LIN {X 0,Y 431.431,Z 392.895,A -85,B 0,C 180,E1 -9540.932,E2 -9540.932} C_VEL
LIN {X 0,Y 431.488,Z 391.643,A -85,B 0,C 180,E1 -9541.866,E2 -9541.866} C_VEL
LIN {X 0,Y 431.805,Z 388.442,A -85,B 0,C 180,E1 -9543.264,E2 -9543.264} C_VEL
LIN {X 0,Y 431.906,Z 385.263,A -85,B 0,C 180,E1 -9544.198,E2 -9544.198} C_VEL
LIN {X 0,Y 432.129,Z 379.971,A -85,B 0,C 180,E1 -9545.365,E2 -9545.365} C_VEL
LIN {X 0,Y 432.279,Z 374.459,A -85,B 0,C 180,E1 -9546.299,E2 -9546.299} C_VEL
LIN {X 0,Y 432.336,Z 367.466,A -85,B 0,C 180,E1 -9547.221,E2 -9547.221} C_VEL
LIN {X 0,Y 432.6,Z 359.724,A -85,B 0,C 180,E1 -9548.018,E2 -9548.018} C_VEL
LIN {X 0,Y 432.755,Z 351.837,A -85,B 0,C 180,E1 -9548.638,E2 -9548.638} C_VEL
LIN {X 0,Y 432.779,Z 343.053,A -85,B 0,C 180,E1 -9549.168,E2 -9549.168} C_VEL
LIN {X 0,Y 431.838,Z 336.706,A -85,B 0,C 180,E1 -9549.483,E2 -9549.483} C_VEL
LIN {X 0,Y 431.977,Z 329.555,A -85,B 0,C 180,E1 -9552.534,E2 -9552.534} C_VEL
LIN {X 0,Y 431.962,Z 320.915,A -85,B 0,C 180,E1 -9556.274,E2 -9556.274} C_VEL
LIN {X 0,Y 432.057,Z 313.809,A -85,B 0,C 180,E1 -9559.36,E2 -9559.36} C_VEL
LIN {X 0,Y 432.075,Z 306.679,A -85,B 0,C 180,E1 -9562.471,E2 -9562.471} C_VEL
LIN {X 0,Y 432.147,Z 299.603,A -85,B 0,C 180,E1 -9565.527,E2 -9565.527} C_VEL
LIN {X 0,Y 432.259,Z 292.542,A -85,B 0,C 180,E1 -9568.601,E2 -9568.601} C_VEL
LIN {X 0,Y 432.354,Z 290.632,A -85,B 0,C 180,E1 -9569.452,E2 -9569.452} C_VEL
LIN {X 0,Y 432.31,Z 290.631,A -85,B 0,C 180,E1 -9572.442,E2 -9572.442} C_VEL
LIN {X 0,Y 432.33,Z 290.629,A -85,B 0,C 180,E1 -9575.817,E2 -9575.817} C_VEL
LIN {X 0,Y 432.323,Z 290.633,A -85,B 0,C 180,E1 -9578.711,E2 -9578.711} C_VEL
LIN {X 0,Y 432.313,Z 290.632,A -85,B 0,C 180,E1 -9581.797,E2 -9581.797} C_VEL
LIN {X 0,Y 432.326,Z 290.632,A -85,B 0,C 180,E1 -9584.346,E2 -9584.346} C_VEL
LIN {X 0,Y 432.312,Z 290.635,A -85,B 0,C 180,E1 -9587.014,E2 -9587.014} C_VEL
LIN {X 0,Y 432.333,Z 290.631,A -85,B 0,C 180,E1 -9589.818,E2 -9589.818} C_VEL
LIN {X 0,Y 432.307,Z 290.634,A -85,B 0,C 180,E1 -9593.022,E2 -9593.022} C_VEL
LIN {X 0,Y 432.35,Z 290.63,A -85,B 0,C 180,E1 -9595.995,E2 -9595.995} C_VEL
LIN {X 0,Y 432.385,Z 290.625,A -85,B 0,C 180,E1 -9599.743,E2 -9599.743} C_VEL
LIN {X 0,Y 432.39,Z 290.625,A -85,B 0,C 180,E1 -9603.371,E2 -9603.371} C_VEL
LIN {X 0,Y 432.36,Z 290.629,A -85,B 0,C 180,E1 -9606.023,E2 -9606.023} C_VEL
LIN {X 0,Y 432.339,Z 290.632,A -85,B 0,C 180,E1 -9609.045,E2 -9609.045} C_VEL
LIN {X 0,Y 432.366,Z 290.627,A -85,B 0,C 180,E1 -9612.011,E2 -9612.011} C_VEL
LIN {X 0,Y 432.383,Z 290.626,A -85,B 0,C 180,E1 -9614.926,E2 -9614.926} C_VEL
LIN {X 0,Y 432.446,Z 290.616,A -85,B 0,C 180,E1 -9617.803,E2 -9617.803} C_VEL
LIN {X 0,Y 432.451,Z 290.615,A -85,B 0,C 180,E1 -9621.589,E2 -9621.589} C_VEL
LIN {X 0,Y 432.567,Z 290.604,A -85,B 0,C 180,E1 -9624.406,E2 -9624.406} C_VEL
LIN {X 0,Y 432.582,Z 290.603,A -85,B 0,C 180,E1 -9628.138,E2 -9628.138} C_VEL
LIN {X 0,Y 432.597,Z 290.601,A -85,B 0,C 180,E1 -9630.119,E2 -9630.119} C_VEL
LIN {X 0,Y 432.548,Z 290.602,A -85,B 0,C 180,E1 -9632.794,E2 -9632.794} C_VEL
LIN {X 0,Y 432.337,Z 290.629,A -85,B 0,C 180,E1 -9634.194,E2 -9634.194} C_VEL
LIN {X 0,Y 431.716,Z 290.706,A -85,B 0,C 180,E1 -9634.973,E2 -9634.973} C_VEL
LIN {X 0,Y 428.929,Z 291.054,A -85,B 0,C 180,E1 -9636.239,E2 -9636.239} C_VEL
LIN {X 0,Y 426.54,Z 291.353,A -85,B 0,C 180,E1 -9637.261,E2 -9637.261} C_VEL
LIN {X 0,Y 425.497,Z 291.483,A -85,B 0,C 180,E1 -9638.049,E2 -9638.049} C_VEL
LIN {X 0,Y 425.404,Z 291.493,A -85,B 0,C 180,E1 -9638.317,E2 -9638.317} C_VEL
LIN {X 0,Y 425.337,Z 291.505,A -85,B 0,C 180,E1 -9641.436,E2 -9641.436} C_VEL
LIN {X 0,Y 425.336,Z 291.503,A -85,B 0,C 180,E1 -9644.35,E2 -9644.35} C_VEL
LIN {X 0,Y 425.33,Z 291.507,A -85,B 0,C 180,E1 -9647.303,E2 -9647.303} C_VEL
LIN {X 0,Y 425.284,Z 291.51,A -85,B 0,C 180,E1 -9650.306,E2 -9650.306} C_VEL
LIN {X 0,Y 425.296,Z 291.509,A -85,B 0,C 180,E1 -9653.366,E2 -9653.366} C_VEL
LIN {X 0,Y 425.338,Z 291.504,A -85,B 0,C 180,E1 -9656.845,E2 -9656.845} C_VEL
LIN {X 0,Y 425.308,Z 291.508,A -85,B 0,C 180,E1 -9659.718,E2 -9659.718} C_VEL
LIN {X 0,Y 425.275,Z 291.511,A -85,B 0,C 180,E1 -9663.049,E2 -9663.049} C_VEL
LIN {X 0,Y 425.276,Z 291.511,A -85,B 0,C 180,E1 -9665.93,E2 -9665.93} C_VEL
LIN {X 0,Y 425.295,Z 291.508,A -85,B 0,C 180,E1 -9669.046,E2 -9669.046} C_VEL
LIN {X 0,Y 425.267,Z 291.511,A -85,B 0,C 180,E1 -9672.654,E2 -9672.654} C_VEL
LIN {X 0,Y 425.253,Z 291.512,A -85,B 0,C 180,E1 -9676.045,E2 -9676.045} C_VEL
LIN {X 0,Y 425.249,Z 291.513,A -85,B 0,C 180,E1 -9678.621,E2 -9678.621} C_VEL
LIN {X 0,Y 425.274,Z 291.513,A -85,B 0,C 180,E1 -9681.101,E2 -9681.101} C_VEL
LIN {X 0,Y 425.288,Z 291.511,A -85,B 0,C 180,E1 -9684.665,E2 -9684.665} C_VEL
LIN {X 0,Y 425.325,Z 291.502,A -85,B 0,C 180,E1 -9688.08,E2 -9688.08} C_VEL
LIN {X 0,Y 425.41,Z 291.557,A -85,B 0,C 180,E1 -9689.302,E2 -9689.302} C_VEL
LIN {X 0,Y 425.439,Z 295.465,A -85,B 0,C 180,E1 -9691.378,E2 -9691.378} C_VEL
LIN {X 0,Y 425.168,Z 301.535,A -85,B 0,C 180,E1 -9694.548,E2 -9694.548} C_VEL
LIN {X 0,Y 424.965,Z 307.922,A -85,B 0,C 180,E1 -9697.838,E2 -9697.838} C_VEL
LIN {X 0,Y 424.857,Z 313.552,A -85,B 0,C 180,E1 -9700.682,E2 -9700.682} C_VEL
LIN {X 0,Y 424.689,Z 319.597,A -85,B 0,C 180,E1 -9703.703,E2 -9703.703} C_VEL
LIN {X 0,Y 424.581,Z 327.506,A -85,B 0,C 180,E1 -9707.586,E2 -9707.586} C_VEL
LIN {X 0,Y 424.422,Z 332.382,A -85,B 0,C 180,E1 -9709.898,E2 -9709.898} C_VEL
LIN {X 0,Y 425.912,Z 342.722,A -85,B 0,C 180,E1 -9710.444,E2 -9710.444} C_VEL
LIN {X 0,Y 426.109,Z 349.157,A -85,B 0,C 180,E1 -9710.867,E2 -9710.867} C_VEL
LIN {X 0,Y 425.799,Z 357.927,A -85,B 0,C 180,E1 -9711.578,E2 -9711.578} C_VEL
LIN {X 0,Y 425.5,Z 365.939,A -85,B 0,C 180,E1 -9712.408,E2 -9712.408} C_VEL
LIN {X 0,Y 425.269,Z 373.188,A -85,B 0,C 180,E1 -9713.358,E2 -9713.358} C_VEL
LIN {X 0,Y 425.072,Z 380.203,A -85,B 0,C 180,E1 -9714.546,E2 -9714.546} C_VEL
LIN {X 0,Y 424.872,Z 385.525,A -85,B 0,C 180,E1 -9715.732,E2 -9715.732} C_VEL
LIN {X 0,Y 424.62,Z 390.099,A -85,B 0,C 180,E1 -9717.155,E2 -9717.155} C_VEL
LIN {X 0,Y 424.439,Z 392.202,A -85,B 0,C 180,E1 -9718.103,E2 -9718.103} C_VEL
LIN {X 0,Y 424.384,Z 393.597,A -85,B 0,C 180,E1 -9719.052,E2 -9719.052} C_VEL
LIN {X 0,Y 424.397,Z 394.313,A -85,B 0,C 180,E1 -9720.001,E2 -9720.001} C_VEL
LIN {X 0,Y 424.439,Z 394.36,A -85,B 0,C 180,E1 -9720.95,E2 -9720.95} C_VEL
LIN {X 0,Y 424.516,Z 393.742,A -85,B 0,C 180,E1 -9721.899,E2 -9721.899} C_VEL
LIN {X 0,Y 424.66,Z 392.447,A -85,B 0,C 180,E1 -9722.847,E2 -9722.847} C_VEL
LIN {X 0,Y 424.926,Z 390.439,A -85,B 0,C 180,E1 -9723.795,E2 -9723.795} C_VEL
LIN {X 0,Y 425.187,Z 387.687,A -85,B 0,C 180,E1 -9724.742,E2 -9724.742} C_VEL
LIN {X 0,Y 425.583,Z 383.077,A -85,B 0,C 180,E1 -9725.925,E2 -9725.925} C_VEL
LIN {X 0,Y 425.972,Z 376.983,A -85,B 0,C 180,E1 -9727.109,E2 -9727.109} C_VEL
LIN {X 0,Y 426.429,Z 369.893,A -85,B 0,C 180,E1 -9728.171,E2 -9728.171} C_VEL
LIN {X 0,Y 426.984,Z 361.78,A -85,B 0,C 180,E1 -9729.116,E2 -9729.116} C_VEL
LIN {X 0,Y 427.458,Z 352.678,A -85,B 0,C 180,E1 -9729.942,E2 -9729.942} C_VEL
LIN {X 0,Y 427.53,Z 347.987,A -85,B 0,C 180,E1 -9730.299,E2 -9730.299} C_VEL
LIN {X 0,Y 425.577,Z 337.921,A -85,B 0,C 180,E1 -9731.009,E2 -9731.009} C_VEL
LIN {X 0,Y 424.97,Z 335.305,A -85,B 0,C 180,E1 -9731.206,E2 -9731.206} C_VEL
LIN {X 0,Y 425.162,Z 331.199,A -85,B 0,C 180,E1 -9733.382,E2 -9733.382} C_VEL
LIN {X 0,Y 425.431,Z 325.231,A -85,B 0,C 180,E1 -9736.635,E2 -9736.635} C_VEL
LIN {X 0,Y 425.776,Z 318.779,A -85,B 0,C 180,E1 -9740.283,E2 -9740.283} C_VEL
LIN {X 0,Y 426.086,Z 313.641,A -85,B 0,C 180,E1 -9743.321,E2 -9743.321} C_VEL
LIN {X 0,Y 426.534,Z 308.597,A -85,B 0,C 180,E1 -9746.417,E2 -9746.417} C_VEL
LIN {X 0,Y 426.992,Z 304.201,A -85,B 0,C 180,E1 -9749.267,E2 -9749.267} C_VEL
LIN {X 0,Y 427.019,Z 301.577,A -85,B 0,C 180,E1 -9751.148,E2 -9751.148} C_VEL
LIN {X 0,Y 426.838,Z 299.371,A -85,B 0,C 180,E1 -9752.913,E2 -9752.913} C_VEL
LIN {X 0,Y 426.407,Z 296.853,A -85,B 0,C 180,E1 -9755.231,E2 -9755.231} C_VEL
LIN {X 0,Y 425.993,Z 294.732,A -85,B 0,C 180,E1 -9757.636,E2 -9757.636} C_VEL
LIN {X 0,Y 425.623,Z 292.959,A -85,B 0,C 180,E1 -9760.574,E2 -9760.574} C_VEL
LIN {X 0,Y 425.422,Z 292.31,A -85,B 0,C 180,E1 -9763.374,E2 -9763.374} C_VEL
LIN {X 0,Y 425.543,Z 292.781,A -85,B 0,C 180,E1 -9766.08,E2 -9766.08} C_VEL
LIN {X 0,Y 425.84,Z 293.804,A -85,B 0,C 180,E1 -9767.961,E2 -9767.961} C_VEL
LIN {X 0,Y 426.327,Z 295.602,A -85,B 0,C 180,E1 -9769.99,E2 -9769.99} C_VEL
LIN {X 0,Y 427.12,Z 298.823,A -85,B 0,C 180,E1 -9772.496,E2 -9772.496} C_VEL
LIN {X 0,Y 428.239,Z 303.443,A -85,B 0,C 180,E1 -9775.143,E2 -9775.143} C_VEL
LIN {X 0,Y 429.35,Z 308.119,A -85,B 0,C 180,E1 -9777.304,E2 -9777.304} C_VEL
LIN {X 0,Y 430.605,Z 314.841,A -85,B 0,C 180,E1 -9779.887,E2 -9779.887} C_VEL
LIN {X 0,Y 430.728,Z 317.29,A -85,B 0,C 180,E1 -9780.692,E2 -9780.692} C_VEL
LIN {X 0,Y 429.254,Z 326.071,A -85,B 0,C 180,E1 -9783.24,E2 -9783.24} C_VEL
LIN {X 0,Y 427.548,Z 339.217,A -85,B 0,C 180,E1 -9786.764,E2 -9786.764} C_VEL
LIN {X 0,Y 426.625,Z 349.188,A -85,B 0,C 180,E1 -9789.257,E2 -9789.257} C_VEL
LIN {X 0,Y 425.685,Z 363.777,A -85,B 0,C 180,E1 -9792.712,E2 -9792.712} C_VEL
LIN {X 0,Y 425.548,Z 366.714,A -85,B 0,C 180,E1 -9793.388,E2 -9793.388} C_VEL
LIN {X 0,Y 427.239,Z 380.58,A -85,B 0,C 180,E1 -9793.883,E2 -9793.883} C_VEL
LIN {X 0,Y 427.862,Z 392.817,A -85,B 0,C 180,E1 -9794.458,E2 -9794.458} C_VEL
LIN {X 0,Y 427.224,Z 405.62,A -85,B 0,C 180,E1 -9795.227,E2 -9795.227} C_VEL
LIN {X 0,Y 426.563,Z 416.33,A -85,B 0,C 180,E1 -9796.057,E2 -9796.057} C_VEL
LIN {X 0,Y 426.089,Z 426.068,A -85,B 0,C 180,E1 -9796.996,E2 -9796.996} C_VEL
LIN {X 0,Y 425.42,Z 435.337,A -85,B 0,C 180,E1 -9798.083,E2 -9798.083} C_VEL
LIN {X 0,Y 424.995,Z 443.71,A -85,B 0,C 180,E1 -9799.278,E2 -9799.278} C_VEL
LIN {X 0,Y 424.666,Z 451.921,A -85,B 0,C 180,E1 -9800.714,E2 -9800.714} C_VEL
LIN {X 0,Y 424.5,Z 457.482,A -85,B 0,C 180,E1 -9801.91,E2 -9801.91} C_VEL
LIN {X 0,Y 424.376,Z 463.56,A -85,B 0,C 180,E1 -9803.544,E2 -9803.544} C_VEL
LIN {X 0,Y 424.29,Z 468.247,A -85,B 0,C 180,E1 -9805.249,E2 -9805.249} C_VEL
LIN {X 0,Y 424.391,Z 470.225,A -85,B 0,C 180,E1 -9806.202,E2 -9806.202} C_VEL
LIN {X 0,Y 424.431,Z 471.7,A -85,B 0,C 180,E1 -9807.153,E2 -9807.153} C_VEL
LIN {X 0,Y 424.379,Z 472.748,A -85,B 0,C 180,E1 -9808.102,E2 -9808.102} C_VEL
LIN {X 0,Y 424.299,Z 473.383,A -85,B 0,C 180,E1 -9809.051,E2 -9809.051} C_VEL
LIN {X 0,Y 424.292,Z 473.558,A -85,B 0,C 180,E1 -9810,E2 -9810} C_VEL
LIN {X 0,Y 424.297,Z 473.314,A -85,B 0,C 180,E1 -9810.949,E2 -9810.949} C_VEL
LIN {X 0,Y 424.378,Z 472.67,A -85,B 0,C 180,E1 -9811.898,E2 -9811.898} C_VEL
LIN {X 0,Y 424.5,Z 471.576,A -85,B 0,C 180,E1 -9812.847,E2 -9812.847} C_VEL
LIN {X 0,Y 424.31,Z 469.054,A -85,B 0,C 180,E1 -9814.275,E2 -9814.275} C_VEL
LIN {X 0,Y 424.379,Z 465.475,A -85,B 0,C 180,E1 -9815.703,E2 -9815.703} C_VEL
LIN {X 0,Y 424.433,Z 460.7,A -85,B 0,C 180,E1 -9817.134,E2 -9817.134} C_VEL
LIN {X 0,Y 424.543,Z 454.589,A -85,B 0,C 180,E1 -9818.568,E2 -9818.568} C_VEL
LIN {X 0,Y 424.774,Z 446.92,A -85,B 0,C 180,E1 -9820.005,E2 -9820.005} C_VEL
LIN {X 0,Y 425.172,Z 438.998,A -85,B 0,C 180,E1 -9821.199,E2 -9821.199} C_VEL
LIN {X 0,Y 425.61,Z 430.347,A -85,B 0,C 180,E1 -9822.275,E2 -9822.275} C_VEL
LIN {X 0,Y 425.952,Z 422.768,A -85,B 0,C 180,E1 -9823.069,E2 -9823.069} C_VEL
LIN {X 0,Y 426.519,Z 411.011,A -85,B 0,C 180,E1 -9824.066,E2 -9824.066} C_VEL
LIN {X 0,Y 427.09,Z 399.322,A -85,B 0,C 180,E1 -9824.838,E2 -9824.838} C_VEL
LIN {X 0,Y 427.203,Z 388.532,A -85,B 0,C 180,E1 -9825.383,E2 -9825.383} C_VEL
LIN {X 0,Y 426,Z 375.127,A -85,B 0,C 180,E1 -9825.888,E2 -9825.888} C_VEL
LIN {X 0,Y 425.312,Z 367.811,A -85,B 0,C 180,E1 -9826.099,E2 -9826.099} C_VEL
LIN {X 0,Y 426.031,Z 354.032,A -85,B 0,C 180,E1 -9829.265,E2 -9829.265} C_VEL
LIN {X 0,Y 427.055,Z 339.899,A -85,B 0,C 180,E1 -9832.553,E2 -9832.553} C_VEL
LIN {X 0,Y 428.279,Z 325.124,A -85,B 0,C 180,E1 -9836.052,E2 -9836.052} C_VEL
LIN {X 0,Y 429.459,Z 312.388,A -85,B 0,C 180,E1 -9839.134,E2 -9839.134} C_VEL
LIN {X 0,Y 428.62,Z 306.988,A -85,B 0,C 180,E1 -9840.551,E2 -9840.551} C_VEL
LIN {X 0,Y 425.673,Z 293.201,A -85,B 0,C 180,E1 -9844.358,E2 -9844.358} C_VEL
LIN {X 0,Y 425.309,Z 291.509,A -85,B 0,C 180,E1 -9844.858,E2 -9844.858} C_VEL
LIN {X 0,Y 425.284,Z 291.512,A -85,B 0,C 180,E1 -9847.694,E2 -9847.694} C_VEL
LIN {X 0,Y 425.285,Z 291.513,A -85,B 0,C 180,E1 -9850.52,E2 -9850.52} C_VEL
LIN {X 0,Y 425.263,Z 291.512,A -85,B 0,C 180,E1 -9853.35,E2 -9853.35} C_VEL
LIN {X 0,Y 425.263,Z 291.512,A -85,B 0,C 180,E1 -9856.649,E2 -9856.649} C_VEL
LIN {X 0,Y 425.295,Z 291.508,A -85,B 0,C 180,E1 -9859.873,E2 -9859.873} C_VEL
LIN {X 0,Y 425.284,Z 291.511,A -85,B 0,C 180,E1 -9862.488,E2 -9862.488} C_VEL
LIN {X 0,Y 425.311,Z 291.511,A -85,B 0,C 180,E1 -9865.817,E2 -9865.817} C_VEL
LIN {X 0,Y 425.288,Z 291.514,A -85,B 0,C 180,E1 -9869.24,E2 -9869.24} C_VEL
LIN {X 0,Y 425.311,Z 291.731,A -85,B 0,C 180,E1 -9870.008,E2 -9870.008} C_VEL
LIN {X 0,Y 425.767,Z 295.291,A -85,B 0,C 180,E1 -9871.399,E2 -9871.399} C_VEL
LIN {X 0,Y 425.635,Z 303.415,A -85,B 0,C 180,E1 -9874.575,E2 -9874.575} C_VEL
LIN {X 0,Y 425.538,Z 312.26,A -85,B 0,C 180,E1 -9878.185,E2 -9878.185} C_VEL
LIN {X 0,Y 425.438,Z 319.451,A -85,B 0,C 180,E1 -9881.207,E2 -9881.207} C_VEL
LIN {X 0,Y 425.368,Z 326.466,A -85,B 0,C 180,E1 -9884.179,E2 -9884.179} C_VEL
LIN {X 0,Y 425.402,Z 335.436,A -85,B 0,C 180,E1 -9888.081,E2 -9888.081} C_VEL
LIN {X 0,Y 425.301,Z 339.67,A -85,B 0,C 180,E1 -9889.917,E2 -9889.917} C_VEL
LIN {X 0,Y 426.723,Z 347.144,A -85,B 0,C 180,E1 -9890.34,E2 -9890.34} C_VEL
LIN {X 0,Y 426.45,Z 356.821,A -85,B 0,C 180,E1 -9890.991,E2 -9890.991} C_VEL
LIN {X 0,Y 426.13,Z 365.402,A -85,B 0,C 180,E1 -9891.785,E2 -9891.785} C_VEL
LIN {X 0,Y 425.771,Z 372.676,A -85,B 0,C 180,E1 -9892.649,E2 -9892.649} C_VEL
LIN {X 0,Y 425.624,Z 378.737,A -85,B 0,C 180,E1 -9893.599,E2 -9893.599} C_VEL
LIN {X 0,Y 425.31,Z 383.556,A -85,B 0,C 180,E1 -9894.547,E2 -9894.547} C_VEL
LIN {X 0,Y 425.194,Z 388.08,A -85,B 0,C 180,E1 -9895.733,E2 -9895.733} C_VEL
LIN {X 0,Y 424.935,Z 390.704,A -85,B 0,C 180,E1 -9896.68,E2 -9896.68} C_VEL
LIN {X 0,Y 424.63,Z 391.791,A -85,B 0,C 180,E1 -9897.153,E2 -9897.153} C_VEL
LIN {X 0,Y 424.489,Z 393.276,A -85,B 0,C 180,E1 -9898.101,E2 -9898.101} C_VEL
LIN {X 0,Y 424.415,Z 394.045,A -85,B 0,C 180,E1 -9899.05,E2 -9899.05} C_VEL
LIN {X 0,Y 424.373,Z 394.123,A -85,B 0,C 180,E1 -9899.999,E2 -9899.999} C_VEL
LIN {X 0,Y 424.368,Z 393.517,A -85,B 0,C 180,E1 -9900.948,E2 -9900.948} C_VEL
LIN {X 0,Y 424.504,Z 391.341,A -85,B 0,C 180,E1 -9902.371,E2 -9902.371} C_VEL
LIN {X 0,Y 424.748,Z 388.935,A -85,B 0,C 180,E1 -9903.319,E2 -9903.319} C_VEL
LIN {X 0,Y 424.981,Z 383.756,A -85,B 0,C 180,E1 -9904.742,E2 -9904.742} C_VEL
LIN {X 0,Y 425.155,Z 377.656,A -85,B 0,C 180,E1 -9905.929,E2 -9905.929} C_VEL
LIN {X 0,Y 425.23,Z 370.847,A -85,B 0,C 180,E1 -9906.95,E2 -9906.95} C_VEL
LIN {X 0,Y 425.455,Z 363.083,A -85,B 0,C 180,E1 -9907.831,E2 -9907.831} C_VEL
LIN {X 0,Y 425.632,Z 355.043,A -85,B 0,C 180,E1 -9908.545,E2 -9908.545} C_VEL
LIN {X 0,Y 425.859,Z 345.965,A -85,B 0,C 180,E1 -9909.138,E2 -9909.138} C_VEL
LIN {X 0,Y 424.8,Z 337.288,A -85,B 0,C 180,E1 -9909.582,E2 -9909.582} C_VEL
LIN {X 0,Y 424.931,Z 330.165,A -85,B 0,C 180,E1 -9912.627,E2 -9912.627} C_VEL
LIN {X 0,Y 424.917,Z 321.461,A -85,B 0,C 180,E1 -9916.401,E2 -9916.401} C_VEL
LIN {X 0,Y 425.025,Z 314.285,A -85,B 0,C 180,E1 -9919.52,E2 -9919.52} C_VEL
LIN {X 0,Y 425.033,Z 306.667,A -85,B 0,C 180,E1 -9922.864,E2 -9922.864} C_VEL
LIN {X 0,Y 425.134,Z 299.493,A -85,B 0,C 180,E1 -9925.98,E2 -9925.98} C_VEL
LIN {X 0,Y 425.335,Z 291.506,A -85,B 0,C 180,E1 -9929.47,E2 -9929.47} C_VEL
LIN {X 0,Y 425.262,Z 291.513,A -85,B 0,C 180,E1 -9933.048,E2 -9933.048} C_VEL
LIN {X 0,Y 425.274,Z 291.508,A -85,B 0,C 180,E1 -9935.927,E2 -9935.927} C_VEL
LIN {X 0,Y 425.258,Z 291.516,A -85,B 0,C 180,E1 -9939.036,E2 -9939.036} C_VEL
LIN {X 0,Y 425.262,Z 291.513,A -85,B 0,C 180,E1 -9942.652,E2 -9942.652} C_VEL
LIN {X 0,Y 425.254,Z 291.512,A -85,B 0,C 180,E1 -9946.043,E2 -9946.043} C_VEL
LIN {X 0,Y 425.267,Z 291.515,A -85,B 0,C 180,E1 -9948.62,E2 -9948.62} C_VEL
LIN {X 0,Y 425.307,Z 291.506,A -85,B 0,C 180,E1 -9951.102,E2 -9951.102} C_VEL
LIN {X 0,Y 425.292,Z 291.509,A -85,B 0,C 180,E1 -9954.663,E2 -9954.663} C_VEL
LIN {X 0,Y 425.263,Z 291.513,A -85,B 0,C 180,E1 -9958.073,E2 -9958.073} C_VEL
LIN {X 0,Y 425.328,Z 291.505,A -85,B 0,C 180,E1 -9961.367,E2 -9961.367} C_VEL
LIN {X 0,Y 425.285,Z 291.51,A -85,B 0,C 180,E1 -9964.554,E2 -9964.554} C_VEL
LIN {X 0,Y 425.277,Z 291.51,A -85,B 0,C 180,E1 -9967.661,E2 -9967.661} C_VEL
LIN {X 0,Y 425.351,Z 291.504,A -85,B 0,C 180,E1 -9970.703,E2 -9970.703} C_VEL
LIN {X 0,Y 425.377,Z 291.498,A -85,B 0,C 180,E1 -9973.688,E2 -9973.688} C_VEL
LIN {X 0,Y 425.399,Z 291.494,A -85,B 0,C 180,E1 -9977.598,E2 -9977.598} C_VEL
LIN {X 0,Y 425.395,Z 291.494,A -85,B 0,C 180,E1 -9981.449,E2 -9981.449} C_VEL
LIN {X 0,Y 425.521,Z 291.483,A -85,B 0,C 180,E1 -9984.313,E2 -9984.313} C_VEL
LIN {X 0,Y 425.552,Z 291.479,A -85,B 0,C 180,E1 -9988.107,E2 -9988.107} C_VEL
LIN {X 0,Y 425.577,Z 291.477,A -85,B 0,C 180,E1 -9990,E2 -9990} C_VEL
LIN {X 0,Y 425.504,Z 291.479,A -85,B 0,C 180,E1 -9992.84,E2 -9992.84} C_VEL
LIN {X 0,Y 425.521,Z 291.483,A -85,B 0,C 180,E1 -9995.687,E2 -9995.687} C_VEL
LIN {X 0,Y 425.404,Z 291.493,A -85,B 0,C 180,E1 -9998.317,E2 -9998.317} C_VEL
LIN {X 0,Y 424.702,Z 291.582,A -85,B 0,C 180,E1 -9999.106,E2 -9999.106} C_VEL
LIN {X 0,Y 421.799,Z 291.942,A -85,B 0,C 180,E1 -10000.389,E2 -10000.389} C_VEL
LIN {X 0,Y 419.386,Z 292.246,A -85,B 0,C 180,E1 -10001.425,E2 -10001.425} C_VEL
LIN {X 0,Y 418.391,Z 292.367,A -85,B 0,C 180,E1 -10002.225,E2 -10002.225} C_VEL
LIN {X 0,Y 418.331,Z 292.374,A -85,B 0,C 180,E1 -10002.496,E2 -10002.496} C_VEL
LIN {X 0,Y 418.29,Z 292.382,A -85,B 0,C 180,E1 -10005.595,E2 -10005.595} C_VEL
LIN {X 0,Y 418.272,Z 292.382,A -85,B 0,C 180,E1 -10008.617,E2 -10008.617} C_VEL
LIN {X 0,Y 418.223,Z 292.389,A -85,B 0,C 180,E1 -10011.697,E2 -10011.697} C_VEL
LIN {X 0,Y 418.273,Z 292.384,A -85,B 0,C 180,E1 -10014.865,E2 -10014.865} C_VEL
LIN {X 0,Y 418.285,Z 292.382,A -85,B 0,C 180,E1 -10018.064,E2 -10018.064} C_VEL
LIN {X 0,Y 418.211,Z 292.391,A -85,B 0,C 180,E1 -10021.396,E2 -10021.396} C_VEL
LIN {X 0,Y 418.257,Z 292.385,A -85,B 0,C 180,E1 -10024.581,E2 -10024.581} C_VEL
LIN {X 0,Y 418.226,Z 292.389,A -85,B 0,C 180,E1 -10027.836,E2 -10027.836} C_VEL
LIN {X 0,Y 418.215,Z 292.39,A -85,B 0,C 180,E1 -10030.949,E2 -10030.949} C_VEL
LIN {X 0,Y 418.202,Z 292.391,A -85,B 0,C 180,E1 -10033.731,E2 -10033.731} C_VEL
LIN {X 0,Y 418.199,Z 292.391,A -85,B 0,C 180,E1 -10036.45,E2 -10036.45} C_VEL
LIN {X 0,Y 418.202,Z 292.394,A -85,B 0,C 180,E1 -10039.134,E2 -10039.134} C_VEL
LIN {X 0,Y 418.231,Z 292.39,A -85,B 0,C 180,E1 -10042.777,E2 -10042.777} C_VEL
LIN {X 0,Y 418.229,Z 292.387,A -85,B 0,C 180,E1 -10046.323,E2 -10046.323} C_VEL
LIN {X 0,Y 418.383,Z 292.437,A -85,B 0,C 180,E1 -10049.249,E2 -10049.249} C_VEL
LIN {X 0,Y 418.411,Z 296.46,A -85,B 0,C 180,E1 -10051.401,E2 -10051.401} C_VEL
LIN {X 0,Y 418.119,Z 302.556,A -85,B 0,C 180,E1 -10054.622,E2 -10054.622} C_VEL
LIN {X 0,Y 417.893,Z 309.625,A -85,B 0,C 180,E1 -10058.287,E2 -10058.287} C_VEL
LIN {X 0,Y 417.719,Z 315.644,A -85,B 0,C 180,E1 -10061.359,E2 -10061.359} C_VEL
LIN {X 0,Y 417.577,Z 321.653,A -85,B 0,C 180,E1 -10064.38,E2 -10064.38} C_VEL
LIN {X 0,Y 417.504,Z 327.987,A -85,B 0,C 180,E1 -10067.512,E2 -10067.512} C_VEL
LIN {X 0,Y 417.384,Z 332.795,A -85,B 0,C 180,E1 -10069.757,E2 -10069.757} C_VEL
LIN {X 0,Y 418.933,Z 343.651,A -85,B 0,C 180,E1 -10070.344,E2 -10070.344} C_VEL
LIN {X 0,Y 419.049,Z 350.807,A -85,B 0,C 180,E1 -10070.833,E2 -10070.833} C_VEL
LIN {X 0,Y 418.701,Z 360.518,A -85,B 0,C 180,E1 -10071.678,E2 -10071.678} C_VEL
LIN {X 0,Y 418.36,Z 369.233,A -85,B 0,C 180,E1 -10072.668,E2 -10072.668} C_VEL
LIN {X 0,Y 418.173,Z 376.491,A -85,B 0,C 180,E1 -10073.73,E2 -10073.73} C_VEL
LIN {X 0,Y 417.976,Z 382.872,A -85,B 0,C 180,E1 -10074.937,E2 -10074.937} C_VEL
LIN {X 0,Y 417.711,Z 387.709,A -85,B 0,C 180,E1 -10076.142,E2 -10076.142} C_VEL
LIN {X 0,Y 417.547,Z 390.617,A -85,B 0,C 180,E1 -10077.107,E2 -10077.107} C_VEL
LIN {X 0,Y 417.385,Z 392.775,A -85,B 0,C 180,E1 -10078.071,E2 -10078.071} C_VEL
LIN {X 0,Y 417.321,Z 394.228,A -85,B 0,C 180,E1 -10079.036,E2 -10079.036} C_VEL
LIN {X 0,Y 417.331,Z 394.998,A -85,B 0,C 180,E1 -10080.001,E2 -10080.001} C_VEL
LIN {X 0,Y 417.38,Z 395.098,A -85,B 0,C 180,E1 -10080.966,E2 -10080.966} C_VEL
LIN {X 0,Y 417.465,Z 394.529,A -85,B 0,C 180,E1 -10081.931,E2 -10081.931} C_VEL
LIN {X 0,Y 417.619,Z 393.285,A -85,B 0,C 180,E1 -10082.895,E2 -10082.895} C_VEL
LIN {X 0,Y 418.182,Z 390.079,A -85,B 0,C 180,E1 -10084.338,E2 -10084.338} C_VEL
LIN {X 0,Y 418.309,Z 387.039,A -85,B 0,C 180,E1 -10085.303,E2 -10085.303} C_VEL
LIN {X 0,Y 418.74,Z 382,A -85,B 0,C 180,E1 -10086.506,E2 -10086.506} C_VEL
LIN {X 0,Y 419.212,Z 375.354,A -85,B 0,C 180,E1 -10087.709,E2 -10087.709} C_VEL
LIN {X 0,Y 419.705,Z 368.559,A -85,B 0,C 180,E1 -10088.669,E2 -10088.669} C_VEL
LIN {X 0,Y 420.316,Z 359.904,A -85,B 0,C 180,E1 -10089.627,E2 -10089.627} C_VEL
LIN {X 0,Y 420.8,Z 350.076,A -85,B 0,C 180,E1 -10090.466,E2 -10090.466} C_VEL
LIN {X 0,Y 419.383,Z 341.712,A -85,B 0,C 180,E1 -10091.112,E2 -10091.112} C_VEL
LIN {X 0,Y 417.995,Z 335.834,A -85,B 0,C 180,E1 -10091.518,E2 -10091.518} C_VEL
LIN {X 0,Y 418.167,Z 331.965,A -85,B 0,C 180,E1 -10093.61,E2 -10093.61} C_VEL
LIN {X 0,Y 418.443,Z 326.227,A -85,B 0,C 180,E1 -10096.793,E2 -10096.793} C_VEL
LIN {X 0,Y 418.777,Z 320.686,A -85,B 0,C 180,E1 -10099.981,E2 -10099.981} C_VEL
LIN {X 0,Y 419.081,Z 316.104,A -85,B 0,C 180,E1 -10102.727,E2 -10102.727} C_VEL
LIN {X 0,Y 419.507,Z 311.197,A -85,B 0,C 180,E1 -10105.823,E2 -10105.823} C_VEL
LIN {X 0,Y 420.078,Z 306.336,A -85,B 0,C 180,E1 -10109.025,E2 -10109.025} C_VEL
LIN {X 0,Y 420.14,Z 303.104,A -85,B 0,C 180,E1 -10111.447,E2 -10111.447} C_VEL
LIN {X 0,Y 419.893,Z 300.675,A -85,B 0,C 180,E1 -10113.529,E2 -10113.529} C_VEL
LIN {X 0,Y 419.454,Z 297.869,A -85,B 0,C 180,E1 -10116.462,E2 -10116.462} C_VEL
LIN {X 0,Y 419.013,Z 295.785,A -85,B 0,C 180,E1 -10119.597,E2 -10119.597} C_VEL
LIN {X 0,Y 418.808,Z 294.887,A -85,B 0,C 180,E1 -10122.408,E2 -10122.408} C_VEL
LIN {X 0,Y 418.845,Z 295.057,A -85,B 0,C 180,E1 -10125.191,E2 -10125.191} C_VEL
LIN {X 0,Y 419.227,Z 296.359,A -85,B 0,C 180,E1 -10127.889,E2 -10127.889} C_VEL
LIN {X 0,Y 419.838,Z 298.756,A -85,B 0,C 180,E1 -10130.497,E2 -10130.497} C_VEL
LIN {X 0,Y 420.792,Z 302.652,A -85,B 0,C 180,E1 -10133.293,E2 -10133.293} C_VEL
LIN {X 0,Y 421.748,Z 306.604,A -85,B 0,C 180,E1 -10135.488,E2 -10135.488} C_VEL
LIN {X 0,Y 422.951,Z 312.007,A -85,B 0,C 180,E1 -10137.936,E2 -10137.936} C_VEL
LIN {X 0,Y 423.927,Z 317.911,A -85,B 0,C 180,E1 -10140.175,E2 -10140.175} C_VEL
LIN {X 0,Y 423.573,Z 321.255,A -85,B 0,C 180,E1 -10141.238,E2 -10141.238} C_VEL
LIN {X 0,Y 421.478,Z 333.704,A -85,B 0,C 180,E1 -10144.836,E2 -10144.836} C_VEL
LIN {X 0,Y 419.979,Z 347.243,A -85,B 0,C 180,E1 -10148.398,E2 -10148.398} C_VEL
LIN {X 0,Y 418.819,Z 361.565,A -85,B 0,C 180,E1 -10151.914,E2 -10151.914} C_VEL
LIN {X 0,Y 418.588,Z 366.57,A -85,B 0,C 180,E1 -10153.073,E2 -10153.073} C_VEL
LIN {X 0,Y 420.337,Z 379.858,A -85,B 0,C 180,E1 -10153.565,E2 -10153.565} C_VEL
LIN {X 0,Y 421.02,Z 392.898,A -85,B 0,C 180,E1 -10154.199,E2 -10154.199} C_VEL
LIN {X 0,Y 420.37,Z 405.488,A -85,B 0,C 180,E1 -10154.981,E2 -10154.981} C_VEL
LIN {X 0,Y 419.636,Z 416.066,A -85,B 0,C 180,E1 -10155.822,E2 -10155.822} C_VEL
LIN {X 0,Y 419.08,Z 426.423,A -85,B 0,C 180,E1 -10156.856,E2 -10156.856} C_VEL
LIN {X 0,Y 418.336,Z 436.715,A -85,B 0,C 180,E1 -10158.124,E2 -10158.124} C_VEL
LIN {X 0,Y 417.867,Z 444.741,A -85,B 0,C 180,E1 -10159.338,E2 -10159.338} C_VEL
LIN {X 0,Y 417.557,Z 452.572,A -85,B 0,C 180,E1 -10160.799,E2 -10160.799} C_VEL
LIN {X 0,Y 417.362,Z 458.86,A -85,B 0,C 180,E1 -10162.258,E2 -10162.258} C_VEL
LIN {X 0,Y 417.273,Z 463.42,A -85,B 0,C 180,E1 -10163.58,E2 -10163.58} C_VEL
LIN {X 0,Y 417.222,Z 467.638,A -85,B 0,C 180,E1 -10165.169,E2 -10165.169} C_VEL
LIN {X 0,Y 417.293,Z 469.593,A -85,B 0,C 180,E1 -10166.137,E2 -10166.137} C_VEL
LIN {X 0,Y 417.355,Z 471.057,A -85,B 0,C 180,E1 -10167.104,E2 -10167.104} C_VEL
LIN {X 0,Y 417.326,Z 472.098,A -85,B 0,C 180,E1 -10168.07,E2 -10168.07} C_VEL
LIN {X 0,Y 417.242,Z 472.713,A -85,B 0,C 180,E1 -10169.035,E2 -10169.035} C_VEL
LIN {X 0,Y 417.231,Z 472.867,A -85,B 0,C 180,E1 -10170,E2 -10170} C_VEL
LIN {X 0,Y 417.24,Z 472.61,A -85,B 0,C 180,E1 -10170.965,E2 -10170.965} C_VEL
LIN {X 0,Y 417.327,Z 471.952,A -85,B 0,C 180,E1 -10171.93,E2 -10171.93} C_VEL
LIN {X 0,Y 417.431,Z 470.821,A -85,B 0,C 180,E1 -10172.895,E2 -10172.895} C_VEL
LIN {X 0,Y 417.244,Z 468.259,A -85,B 0,C 180,E1 -10174.347,E2 -10174.347} C_VEL
LIN {X 0,Y 417.297,Z 464.631,A -85,B 0,C 180,E1 -10175.8,E2 -10175.8} C_VEL
LIN {X 0,Y 417.358,Z 459.8,A -85,B 0,C 180,E1 -10177.256,E2 -10177.256} C_VEL
LIN {X 0,Y 417.478,Z 453.623,A -85,B 0,C 180,E1 -10178.714,E2 -10178.714} C_VEL
LIN {X 0,Y 417.715,Z 445.835,A -85,B 0,C 180,E1 -10180.175,E2 -10180.175} C_VEL
LIN {X 0,Y 418.162,Z 437.807,A -85,B 0,C 180,E1 -10181.39,E2 -10181.39} C_VEL
LIN {X 0,Y 418.667,Z 429.038,A -85,B 0,C 180,E1 -10182.482,E2 -10182.482} C_VEL
LIN {X 0,Y 419.14,Z 418.234,A -85,B 0,C 180,E1 -10183.577,E2 -10183.577} C_VEL
LIN {X 0,Y 419.641,Z 407.646,A -85,B 0,C 180,E1 -10184.426,E2 -10184.426} C_VEL
LIN {X 0,Y 420.234,Z 394.959,A -85,B 0,C 180,E1 -10185.21,E2 -10185.21} C_VEL
LIN {X 0,Y 420.049,Z 387.197,A -85,B 0,C 180,E1 -10185.59,E2 -10185.59} C_VEL
LIN {X 0,Y 418.787,Z 373.339,A -85,B 0,C 180,E1 -10186.107,E2 -10186.107} C_VEL
LIN {X 0,Y 418.298,Z 367.524,A -85,B 0,C 180,E1 -10186.283,E2 -10186.283} C_VEL
LIN {X 0,Y 418.972,Z 354.473,A -85,B 0,C 180,E1 -10189.347,E2 -10189.347} C_VEL
LIN {X 0,Y 420.032,Z 340.656,A -85,B 0,C 180,E1 -10192.634,E2 -10192.634} C_VEL
LIN {X 0,Y 421.333,Z 325.789,A -85,B 0,C 180,E1 -10196.234,E2 -10196.234} C_VEL
LIN {X 0,Y 422.498,Z 314.092,A -85,B 0,C 180,E1 -10199.115,E2 -10199.115} C_VEL
LIN {X 0,Y 421.744,Z 308.699,A -85,B 0,C 180,E1 -10200.547,E2 -10200.547} C_VEL
LIN {X 0,Y 419.006,Z 296.002,A -85,B 0,C 180,E1 -10204.109,E2 -10204.109} C_VEL
LIN {X 0,Y 418.286,Z 292.384,A -85,B 0,C 180,E1 -10205.206,E2 -10205.206} C_VEL
LIN {X 0,Y 418.259,Z 292.388,A -85,B 0,C 180,E1 -10208.441,E2 -10208.441} C_VEL
LIN {X 0,Y 418.227,Z 292.389,A -85,B 0,C 180,E1 -10210.948,E2 -10210.948} C_VEL
LIN {X 0,Y 418.215,Z 292.392,A -85,B 0,C 180,E1 -10213.729,E2 -10213.729} C_VEL
LIN {X 0,Y 418.214,Z 292.39,A -85,B 0,C 180,E1 -10216.448,E2 -10216.448} C_VEL
LIN {X 0,Y 418.229,Z 292.391,A -85,B 0,C 180,E1 -10219.13,E2 -10219.13} C_VEL
LIN {X 0,Y 418.234,Z 292.39,A -85,B 0,C 180,E1 -10222.166,E2 -10222.166} C_VEL
LIN {X 0,Y 418.269,Z 292.388,A -85,B 0,C 180,E1 -10225.419,E2 -10225.419} C_VEL
LIN {X 0,Y 418.212,Z 292.397,A -85,B 0,C 180,E1 -10228.603,E2 -10228.603} C_VEL
LIN {X 0,Y 418.294,Z 292.572,A -85,B 0,C 180,E1 -10229.61,E2 -10229.61} C_VEL
LIN {X 0,Y 418.852,Z 297.098,A -85,B 0,C 180,E1 -10231.431,E2 -10231.431} C_VEL
LIN {X 0,Y 418.705,Z 305.212,A -85,B 0,C 180,E1 -10234.644,E2 -10234.644} C_VEL
LIN {X 0,Y 418.578,Z 312.933,A -85,B 0,C 180,E1 -10237.874,E2 -10237.874} C_VEL
LIN {X 0,Y 418.52,Z 318.946,A -85,B 0,C 180,E1 -10240.375,E2 -10240.375} C_VEL
LIN {X 0,Y 418.413,Z 327.224,A -85,B 0,C 180,E1 -10243.909,E2 -10243.909} C_VEL
LIN {X 0,Y 418.411,Z 335.195,A -85,B 0,C 180,E1 -10247.386,E2 -10247.386} C_VEL
LIN {X 0,Y 418.304,Z 340.378,A -85,B 0,C 180,E1 -10249.655,E2 -10249.655} C_VEL
LIN {X 0,Y 419.897,Z 348.098,A -85,B 0,C 180,E1 -10250.12,E2 -10250.12} C_VEL
LIN {X 0,Y 419.6,Z 356.933,A -85,B 0,C 180,E1 -10250.722,E2 -10250.722} C_VEL
LIN {X 0,Y 419.344,Z 364.721,A -85,B 0,C 180,E1 -10251.423,E2 -10251.423} C_VEL
LIN {X 0,Y 418.897,Z 372.092,A -85,B 0,C 180,E1 -10252.285,E2 -10252.285} C_VEL
LIN {X 0,Y 418.678,Z 378.511,A -85,B 0,C 180,E1 -10253.251,E2 -10253.251} C_VEL
LIN {X 0,Y 418.314,Z 384.558,A -85,B 0,C 180,E1 -10254.455,E2 -10254.455} C_VEL
LIN {X 0,Y 418.174,Z 388.967,A -85,B 0,C 180,E1 -10255.661,E2 -10255.661} C_VEL
LIN {X 0,Y 417.904,Z 391.542,A -85,B 0,C 180,E1 -10256.624,E2 -10256.624} C_VEL
LIN {X 0,Y 417.589,Z 392.613,A -85,B 0,C 180,E1 -10257.105,E2 -10257.105} C_VEL
LIN {X 0,Y 417.435,Z 394.045,A -85,B 0,C 180,E1 -10258.069,E2 -10258.069} C_VEL
LIN {X 0,Y 417.353,Z 394.762,A -85,B 0,C 180,E1 -10259.034,E2 -10259.034} C_VEL
LIN {X 0,Y 417.307,Z 394.793,A -85,B 0,C 180,E1 -10259.999,E2 -10259.999} C_VEL
LIN {X 0,Y 417.306,Z 394.138,A -85,B 0,C 180,E1 -10260.964,E2 -10260.964} C_VEL
LIN {X 0,Y 417.449,Z 391.884,A -85,B 0,C 180,E1 -10262.411,E2 -10262.411} C_VEL
LIN {X 0,Y 417.693,Z 389.401,A -85,B 0,C 180,E1 -10263.375,E2 -10263.375} C_VEL
LIN {X 0,Y 417.935,Z 384.128,A -85,B 0,C 180,E1 -10264.822,E2 -10264.822} C_VEL
LIN {X 0,Y 418.018,Z 379.307,A -85,B 0,C 180,E1 -10265.788,E2 -10265.788} C_VEL
LIN {X 0,Y 418.137,Z 373.217,A -85,B 0,C 180,E1 -10266.755,E2 -10266.755} C_VEL
LIN {X 0,Y 418.332,Z 365.356,A -85,B 0,C 180,E1 -10267.723,E2 -10267.723} C_VEL
LIN {X 0,Y 418.562,Z 357.748,A -85,B 0,C 180,E1 -10268.447,E2 -10268.447} C_VEL
LIN {X 0,Y 418.791,Z 348.472,A -85,B 0,C 180,E1 -10269.111,E2 -10269.111} C_VEL
LIN {X 0,Y 418.664,Z 344.259,A -85,B 0,C 180,E1 -10269.358,E2 -10269.358} C_VEL
LIN {X 0,Y 417.767,Z 337.852,A -85,B 0,C 180,E1 -10269.683,E2 -10269.683} C_VEL
LIN {X 0,Y 417.822,Z 329.843,A -85,B 0,C 180,E1 -10273.123,E2 -10273.123} C_VEL
LIN {X 0,Y 417.859,Z 321.803,A -85,B 0,C 180,E1 -10276.613,E2 -10276.613} C_VEL
LIN {X 0,Y 417.952,Z 313.673,A -85,B 0,C 180,E1 -10280.162,E2 -10280.162} C_VEL
LIN {X 0,Y 418.022,Z 305.38,A -85,B 0,C 180,E1 -10283.796,E2 -10283.796} C_VEL
LIN {X 0,Y 418.146,Z 298.071,A -85,B 0,C 180,E1 -10287.026,E2 -10287.026} C_VEL
LIN {X 0,Y 418.288,Z 292.383,A -85,B 0,C 180,E1 -10289.503,E2 -10289.503} C_VEL
LIN {X 0,Y 418.243,Z 292.386,A -85,B 0,C 180,E1 -10292.84,E2 -10292.84} C_VEL
LIN {X 0,Y 418.237,Z 292.384,A -85,B 0,C 180,E1 -10296.236,E2 -10296.236} C_VEL
LIN {X 0,Y 418.203,Z 292.39,A -85,B 0,C 180,E1 -10299.685,E2 -10299.685} C_VEL
LIN {X 0,Y 418.214,Z 292.389,A -85,B 0,C 180,E1 -10302.318,E2 -10302.318} C_VEL
LIN {X 0,Y 418.228,Z 292.389,A -85,B 0,C 180,E1 -10305.107,E2 -10305.107} C_VEL
LIN {X 0,Y 418.232,Z 292.387,A -85,B 0,C 180,E1 -10307.766,E2 -10307.766} C_VEL
LIN {X 0,Y 418.251,Z 292.388,A -85,B 0,C 180,E1 -10310.617,E2 -10310.617} C_VEL
LIN {X 0,Y 418.237,Z 292.387,A -85,B 0,C 180,E1 -10313.975,E2 -10313.975} C_VEL
LIN {X 0,Y 418.251,Z 292.386,A -85,B 0,C 180,E1 -10317.154,E2 -10317.154} C_VEL
LIN {X 0,Y 418.265,Z 292.384,A -85,B 0,C 180,E1 -10320.838,E2 -10320.838} C_VEL
LIN {X 0,Y 418.261,Z 292.386,A -85,B 0,C 180,E1 -10324.095,E2 -10324.095} C_VEL
LIN {X 0,Y 418.227,Z 292.389,A -85,B 0,C 180,E1 -10327.263,E2 -10327.263} C_VEL
LIN {X 0,Y 418.272,Z 292.383,A -85,B 0,C 180,E1 -10330.364,E2 -10330.364} C_VEL
LIN {X 0,Y 418.305,Z 292.378,A -85,B 0,C 180,E1 -10333.404,E2 -10333.404} C_VEL
LIN {X 0,Y 418.334,Z 292.375,A -85,B 0,C 180,E1 -10336.999,E2 -10336.999} C_VEL
LIN {X 0,Y 418.326,Z 292.379,A -85,B 0,C 180,E1 -10340.328,E2 -10340.328} C_VEL
LIN {X 0,Y 418.433,Z 292.361,A -85,B 0,C 180,E1 -10343.248,E2 -10343.248} C_VEL
LIN {X 0,Y 418.312,Z 292.375,A -85,B 0,C 180,E1 -10345.181,E2 -10345.181} C_VEL
LIN {X 0,Y 418.521,Z 292.356,A -85,B 0,C 180,E1 -10348.075,E2 -10348.075} C_VEL
LIN {X 0,Y 418.529,Z 292.355,A -85,B 0,C 180,E1 -10350,E2 -10350} C_VEL
LIN {X 0,Y 418.461,Z 292.357,A -85,B 0,C 180,E1 -10352.888,E2 -10352.888} C_VEL
LIN {X 0,Y 418.478,Z 292.361,A -85,B 0,C 180,E1 -10355.783,E2 -10355.783} C_VEL
LIN {X 0,Y 418.365,Z 292.37,A -85,B 0,C 180,E1 -10358.696,E2 -10358.696} C_VEL
LIN {X 0,Y 418.302,Z 292.382,A -85,B 0,C 180,E1 -10361.631,E2 -10361.631} C_VEL
LIN {X 0,Y 418.331,Z 292.374,A -85,B 0,C 180,E1 -10362.496,E2 -10362.496} C_VEL
LIN {X 0,Y 417.705,Z 292.455,A -85,B 0,C 180,E1 -10363.3,E2 -10363.3} C_VEL
LIN {X 0,Y 414.813,Z 292.813,A -85,B 0,C 180,E1 -10364.604,E2 -10364.604} C_VEL
LIN {X 0,Y 412.349,Z 293.122,A -85,B 0,C 180,E1 -10365.657,E2 -10365.657} C_VEL
LIN {X 0,Y 411.314,Z 293.249,A -85,B 0,C 180,E1 -10366.472,E2 -10366.472} C_VEL
LIN {X 0,Y 411.244,Z 293.257,A -85,B 0,C 180,E1 -10366.748,E2 -10366.748} C_VEL
LIN {X 0,Y 411.219,Z 293.262,A -85,B 0,C 180,E1 -10369.987,E2 -10369.987} C_VEL
LIN {X 0,Y 411.192,Z 293.267,A -85,B 0,C 180,E1 -10373.148,E2 -10373.148} C_VEL
LIN {X 0,Y 411.228,Z 293.26,A -85,B 0,C 180,E1 -10376.382,E2 -10376.382} C_VEL
LIN {X 0,Y 411.201,Z 293.266,A -85,B 0,C 180,E1 -10379.713,E2 -10379.713} C_VEL
LIN {X 0,Y 411.197,Z 293.265,A -85,B 0,C 180,E1 -10383.157,E2 -10383.157} C_VEL
LIN {X 0,Y 411.187,Z 293.266,A -85,B 0,C 180,E1 -10386.554,E2 -10386.554} C_VEL
LIN {X 0,Y 411.21,Z 293.263,A -85,B 0,C 180,E1 -10389.73,E2 -10389.73} C_VEL
LIN {X 0,Y 411.165,Z 293.27,A -85,B 0,C 180,E1 -10393.135,E2 -10393.135} C_VEL
LIN {X 0,Y 411.159,Z 293.267,A -85,B 0,C 180,E1 -10395.883,E2 -10395.883} C_VEL
LIN {X 0,Y 411.145,Z 293.272,A -85,B 0,C 180,E1 -10398.775,E2 -10398.775} C_VEL
LIN {X 0,Y 411.179,Z 293.264,A -85,B 0,C 180,E1 -10402.027,E2 -10402.027} C_VEL
LIN {X 0,Y 411.197,Z 293.264,A -85,B 0,C 180,E1 -10405.125,E2 -10405.125} C_VEL
LIN {X 0,Y 411.342,Z 293.278,A -85,B 0,C 180,E1 -10409.167,E2 -10409.167} C_VEL
LIN {X 0,Y 411.382,Z 297.417,A -85,B 0,C 180,E1 -10411.424,E2 -10411.424} C_VEL
LIN {X 0,Y 411.032,Z 304.113,A -85,B 0,C 180,E1 -10414.988,E2 -10414.988} C_VEL
LIN {X 0,Y 410.832,Z 310.691,A -85,B 0,C 180,E1 -10418.422,E2 -10418.422} C_VEL
LIN {X 0,Y 410.654,Z 316.758,A -85,B 0,C 180,E1 -10421.543,E2 -10421.543} C_VEL
LIN {X 0,Y 410.49,Z 322.812,A -85,B 0,C 180,E1 -10424.612,E2 -10424.612} C_VEL
LIN {X 0,Y 410.383,Z 329.885,A -85,B 0,C 180,E1 -10428.142,E2 -10428.142} C_VEL
LIN {X 0,Y 410.316,Z 333.065,A -85,B 0,C 180,E1 -10429.609,E2 -10429.609} C_VEL
LIN {X 0,Y 411.78,Z 343.404,A -85,B 0,C 180,E1 -10430.174,E2 -10430.174} C_VEL
LIN {X 0,Y 412.091,Z 349.007,A -85,B 0,C 180,E1 -10430.554,E2 -10430.554} C_VEL
LIN {X 0,Y 411.761,Z 358,A -85,B 0,C 180,E1 -10431.289,E2 -10431.289} C_VEL
LIN {X 0,Y 411.381,Z 367.08,A -85,B 0,C 180,E1 -10432.252,E2 -10432.252} C_VEL
LIN {X 0,Y 411.138,Z 375.232,A -85,B 0,C 180,E1 -10433.376,E2 -10433.376} C_VEL
LIN {X 0,Y 410.969,Z 382.082,A -85,B 0,C 180,E1 -10434.604,E2 -10434.604} C_VEL
LIN {X 0,Y 410.764,Z 386.371,A -85,B 0,C 180,E1 -10435.586,E2 -10435.586} C_VEL
LIN {X 0,Y 410.648,Z 389.743,A -85,B 0,C 180,E1 -10436.567,E2 -10436.567} C_VEL
LIN {X 0,Y 410.333,Z 393.351,A -85,B 0,C 180,E1 -10438.038,E2 -10438.038} C_VEL
LIN {X 0,Y 410.261,Z 394.858,A -85,B 0,C 180,E1 -10439.02,E2 -10439.02} C_VEL
LIN {X 0,Y 410.267,Z 395.684,A -85,B 0,C 180,E1 -10440.001,E2 -10440.001} C_VEL
LIN {X 0,Y 410.321,Z 395.843,A -85,B 0,C 180,E1 -10440.983,E2 -10440.983} C_VEL
LIN {X 0,Y 410.416,Z 395.34,A -85,B 0,C 180,E1 -10441.964,E2 -10441.964} C_VEL
LIN {X 0,Y 410.584,Z 394.166,A -85,B 0,C 180,E1 -10442.945,E2 -10442.945} C_VEL
LIN {X 0,Y 411.166,Z 391.06,A -85,B 0,C 180,E1 -10444.413,E2 -10444.413} C_VEL
LIN {X 0,Y 411.331,Z 388.086,A -85,B 0,C 180,E1 -10445.393,E2 -10445.393} C_VEL
LIN {X 0,Y 411.8,Z 383.162,A -85,B 0,C 180,E1 -10446.616,E2 -10446.616} C_VEL
LIN {X 0,Y 412.291,Z 376.658,A -85,B 0,C 180,E1 -10447.839,E2 -10447.839} C_VEL
LIN {X 0,Y 412.827,Z 370.059,A -85,B 0,C 180,E1 -10448.815,E2 -10448.815} C_VEL
LIN {X 0,Y 413.493,Z 361.742,A -85,B 0,C 180,E1 -10449.787,E2 -10449.787} C_VEL
LIN {X 0,Y 414.055,Z 352.419,A -85,B 0,C 180,E1 -10450.638,E2 -10450.638} C_VEL
LIN {X 0,Y 413.308,Z 346.152,A -85,B 0,C 180,E1 -10451.154,E2 -10451.154} C_VEL
LIN {X 0,Y 411.006,Z 336.285,A -85,B 0,C 180,E1 -10451.905,E2 -10451.905} C_VEL
LIN {X 0,Y 411.269,Z 330.965,A -85,B 0,C 180,E1 -10454.853,E2 -10454.853} C_VEL
LIN {X 0,Y 411.561,Z 325.654,A -85,B 0,C 180,E1 -10457.902,E2 -10457.902} C_VEL
LIN {X 0,Y 411.904,Z 320.458,A -85,B 0,C 180,E1 -10460.997,E2 -10460.997} C_VEL
LIN {X 0,Y 412.333,Z 315.395,A -85,B 0,C 180,E1 -10464.147,E2 -10464.147} C_VEL
LIN {X 0,Y 412.973,Z 309.986,A -85,B 0,C 180,E1 -10467.755,E2 -10467.755} C_VEL
LIN {X 0,Y 413.289,Z 307.035,A -85,B 0,C 180,E1 -10469.858,E2 -10469.858} C_VEL
LIN {X 0,Y 413.264,Z 304.617,A -85,B 0,C 180,E1 -10471.817,E2 -10471.817} C_VEL
LIN {X 0,Y 413.017,Z 302.094,A -85,B 0,C 180,E1 -10474.163,E2 -10474.163} C_VEL
LIN {X 0,Y 412.658,Z 299.786,A -85,B 0,C 180,E1 -10476.826,E2 -10476.826} C_VEL
LIN {X 0,Y 412.283,Z 298.019,A -85,B 0,C 180,E1 -10479.906,E2 -10479.906} C_VEL
LIN {X 0,Y 412.134,Z 297.327,A -85,B 0,C 180,E1 -10483.01,E2 -10483.01} C_VEL
LIN {X 0,Y 412.272,Z 297.811,A -85,B 0,C 180,E1 -10485.724,E2 -10485.724} C_VEL
LIN {X 0,Y 412.737,Z 299.441,A -85,B 0,C 180,E1 -10488.524,E2 -10488.524} C_VEL
LIN {X 0,Y 413.374,Z 301.982,A -85,B 0,C 180,E1 -10491.019,E2 -10491.019} C_VEL
LIN {X 0,Y 414.27,Z 305.639,A -85,B 0,C 180,E1 -10493.575,E2 -10493.575} C_VEL
LIN {X 0,Y 415.361,Z 310.199,A -85,B 0,C 180,E1 -10496.057,E2 -10496.057} C_VEL
LIN {X 0,Y 416.501,Z 315.646,A -85,B 0,C 180,E1 -10498.46,E2 -10498.46} C_VEL
LIN {X 0,Y 417.135,Z 320.226,A -85,B 0,C 180,E1 -10500.197,E2 -10500.197} C_VEL
LIN {X 0,Y 416.284,Z 325.196,A -85,B 0,C 180,E1 -10501.789,E2 -10501.789} C_VEL
LIN {X 0,Y 414.499,Z 335.92,A -85,B 0,C 180,E1 -10504.92,E2 -10504.92} C_VEL
LIN {X 0,Y 412.928,Z 349.308,A -85,B 0,C 180,E1 -10508.535,E2 -10508.535} C_VEL
LIN {X 0,Y 411.753,Z 363.562,A -85,B 0,C 180,E1 -10512.107,E2 -10512.107} C_VEL
LIN {X 0,Y 411.618,Z 366.159,A -85,B 0,C 180,E1 -10512.718,E2 -10512.718} C_VEL
LIN {X 0,Y 413.386,Z 378.627,A -85,B 0,C 180,E1 -10513.201,E2 -10513.201} C_VEL
LIN {X 0,Y 414.169,Z 392.046,A -85,B 0,C 180,E1 -10513.867,E2 -10513.867} C_VEL
LIN {X 0,Y 413.622,Z 403.77,A -85,B 0,C 180,E1 -10514.604,E2 -10514.604} C_VEL
LIN {X 0,Y 412.727,Z 415.899,A -85,B 0,C 180,E1 -10515.579,E2 -10515.579} C_VEL
LIN {X 0,Y 412.078,Z 426.82,A -85,B 0,C 180,E1 -10516.709,E2 -10516.709} C_VEL
LIN {X 0,Y 411.344,Z 436.342,A -85,B 0,C 180,E1 -10517.919,E2 -10517.919} C_VEL
LIN {X 0,Y 410.857,Z 444.301,A -85,B 0,C 180,E1 -10519.154,E2 -10519.154} C_VEL
LIN {X 0,Y 410.514,Z 452.077,A -85,B 0,C 180,E1 -10520.64,E2 -10520.64} C_VEL
LIN {X 0,Y 410.289,Z 458.323,A -85,B 0,C 180,E1 -10522.124,E2 -10522.124} C_VEL
LIN {X 0,Y 410.202,Z 463.184,A -85,B 0,C 180,E1 -10523.579,E2 -10523.579} C_VEL
LIN {X 0,Y 410.158,Z 467.045,A -85,B 0,C 180,E1 -10525.085,E2 -10525.085} C_VEL
LIN {X 0,Y 410.198,Z 468.966,A -85,B 0,C 180,E1 -10526.07,E2 -10526.07} C_VEL
LIN {X 0,Y 410.28,Z 470.419,A -85,B 0,C 180,E1 -10527.054,E2 -10527.054} C_VEL
LIN {X 0,Y 410.275,Z 471.449,A -85,B 0,C 180,E1 -10528.037,E2 -10528.037} C_VEL
LIN {X 0,Y 410.187,Z 472.036,A -85,B 0,C 180,E1 -10529.018,E2 -10529.018} C_VEL
LIN {X 0,Y 410.172,Z 472.172,A -85,B 0,C 180,E1 -10530,E2 -10530} C_VEL
LIN {X 0,Y 410.184,Z 471.9,A -85,B 0,C 180,E1 -10530.982,E2 -10530.982} C_VEL
LIN {X 0,Y 410.278,Z 471.218,A -85,B 0,C 180,E1 -10531.963,E2 -10531.963} C_VEL
LIN {X 0,Y 410.365,Z 470.055,A -85,B 0,C 180,E1 -10532.945,E2 -10532.945} C_VEL
LIN {X 0,Y 410.181,Z 467.448,A -85,B 0,C 180,E1 -10534.422,E2 -10534.422} C_VEL
LIN {X 0,Y 410.223,Z 463.767,A -85,B 0,C 180,E1 -10535.9,E2 -10535.9} C_VEL
LIN {X 0,Y 410.283,Z 458.875,A -85,B 0,C 180,E1 -10537.381,E2 -10537.381} C_VEL
LIN {X 0,Y 410.42,Z 452.629,A -85,B 0,C 180,E1 -10538.866,E2 -10538.866} C_VEL
LIN {X 0,Y 410.68,Z 444.713,A -85,B 0,C 180,E1 -10540.352,E2 -10540.352} C_VEL
LIN {X 0,Y 411.141,Z 436.578,A -85,B 0,C 180,E1 -10541.587,E2 -10541.587} C_VEL
LIN {X 0,Y 411.73,Z 427.691,A -85,B 0,C 180,E1 -10542.696,E2 -10542.696} C_VEL
LIN {X 0,Y 412.109,Z 417.668,A -85,B 0,C 180,E1 -10543.719,E2 -10543.719} C_VEL
LIN {X 0,Y 412.676,Z 405.761,A -85,B 0,C 180,E1 -10544.674,E2 -10544.674} C_VEL
LIN {X 0,Y 413.237,Z 393.822,A -85,B 0,C 180,E1 -10545.411,E2 -10545.411} C_VEL
LIN {X 0,Y 412.59,Z 382.178,A -85,B 0,C 180,E1 -10545.958,E2 -10545.958} C_VEL
LIN {X 0,Y 411.333,Z 368.937,A -85,B 0,C 180,E1 -10546.391,E2 -10546.391} C_VEL
LIN {X 0,Y 411.259,Z 367.345,A -85,B 0,C 180,E1 -10546.442,E2 -10546.442} C_VEL
LIN {X 0,Y 411.938,Z 354.904,A -85,B 0,C 180,E1 -10549.432,E2 -10549.432} C_VEL
LIN {X 0,Y 413.024,Z 341.14,A -85,B 0,C 180,E1 -10552.775,E2 -10552.775} C_VEL
LIN {X 0,Y 414.397,Z 326.341,A -85,B 0,C 180,E1 -10556.436,E2 -10556.436} C_VEL
LIN {X 0,Y 415.56,Z 314.704,A -85,B 0,C 180,E1 -10559.37,E2 -10559.37} C_VEL
LIN {X 0,Y 414.138,Z 307.146,A -85,B 0,C 180,E1 -10561.455,E2 -10561.455} C_VEL
LIN {X 0,Y 411.586,Z 295.054,A -85,B 0,C 180,E1 -10564.952,E2 -10564.952} C_VEL
LIN {X 0,Y 411.239,Z 293.261,A -85,B 0,C 180,E1 -10565.525,E2 -10565.525} C_VEL
LIN {X 0,Y 411.222,Z 293.262,A -85,B 0,C 180,E1 -10569.224,E2 -10569.224} C_VEL
LIN {X 0,Y 411.187,Z 293.267,A -85,B 0,C 180,E1 -10572.695,E2 -10572.695} C_VEL
LIN {X 0,Y 411.173,Z 293.27,A -85,B 0,C 180,E1 -10575.881,E2 -10575.881} C_VEL
LIN {X 0,Y 411.169,Z 293.269,A -85,B 0,C 180,E1 -10578.771,E2 -10578.771} C_VEL
LIN {X 0,Y 411.212,Z 293.265,A -85,B 0,C 180,E1 -10581.831,E2 -10581.831} C_VEL
LIN {X 0,Y 411.215,Z 293.265,A -85,B 0,C 180,E1 -10585.121,E2 -10585.121} C_VEL
LIN {X 0,Y 411.168,Z 293.275,A -85,B 0,C 180,E1 -10588.002,E2 -10588.002} C_VEL
LIN {X 0,Y 411.226,Z 293.406,A -85,B 0,C 180,E1 -10589.154,E2 -10589.154} C_VEL
LIN {X 0,Y 411.907,Z 297.848,A -85,B 0,C 180,E1 -10590.988,E2 -10590.988} C_VEL
LIN {X 0,Y 411.853,Z 304.508,A -85,B 0,C 180,E1 -10593.66,E2 -10593.66} C_VEL
LIN {X 0,Y 411.723,Z 313.01,A -85,B 0,C 180,E1 -10597.186,E2 -10597.186} C_VEL
LIN {X 0,Y 411.594,Z 319.592,A -85,B 0,C 180,E1 -10600.031,E2 -10600.031} C_VEL
LIN {X 0,Y 411.477,Z 326.853,A -85,B 0,C 180,E1 -10603.119,E2 -10603.119} C_VEL
LIN {X 0,Y 411.41,Z 335.34,A -85,B 0,C 180,E1 -10606.835,E2 -10606.835} C_VEL
LIN {X 0,Y 411.384,Z 341.338,A -85,B 0,C 180,E1 -10609.416,E2 -10609.416} C_VEL
LIN {X 0,Y 413.053,Z 350.013,A -85,B 0,C 180,E1 -10609.955,E2 -10609.955} C_VEL
LIN {X 0,Y 412.746,Z 358.61,A -85,B 0,C 180,E1 -10610.566,E2 -10610.566} C_VEL
LIN {X 0,Y 412.33,Z 367.488,A -85,B 0,C 180,E1 -10611.428,E2 -10611.428} C_VEL
LIN {X 0,Y 411.98,Z 373.385,A -85,B 0,C 180,E1 -10612.155,E2 -10612.155} C_VEL
LIN {X 0,Y 411.724,Z 379.649,A -85,B 0,C 180,E1 -10613.136,E2 -10613.136} C_VEL
LIN {X 0,Y 411.343,Z 385.626,A -85,B 0,C 180,E1 -10614.361,E2 -10614.361} C_VEL
LIN {X 0,Y 411.156,Z 389.92,A -85,B 0,C 180,E1 -10615.587,E2 -10615.587} C_VEL
LIN {X 0,Y 410.87,Z 391.343,A -85,B 0,C 180,E1 -10616.075,E2 -10616.075} C_VEL
LIN {X 0,Y 410.551,Z 393.468,A -85,B 0,C 180,E1 -10617.055,E2 -10617.055} C_VEL
LIN {X 0,Y 410.383,Z 394.827,A -85,B 0,C 180,E1 -10618.036,E2 -10618.036} C_VEL
LIN {X 0,Y 410.291,Z 395.485,A -85,B 0,C 180,E1 -10619.017,E2 -10619.017} C_VEL
LIN {X 0,Y 410.244,Z 395.461,A -85,B 0,C 180,E1 -10619.999,E2 -10619.999} C_VEL
LIN {X 0,Y 410.247,Z 394.751,A -85,B 0,C 180,E1 -10620.98,E2 -10620.98} C_VEL
LIN {X 0,Y 410.396,Z 392.417,A -85,B 0,C 180,E1 -10622.452,E2 -10622.452} C_VEL
LIN {X 0,Y 410.64,Z 389.86,A -85,B 0,C 180,E1 -10623.433,E2 -10623.433} C_VEL
LIN {X 0,Y 410.745,Z 386.474,A -85,B 0,C 180,E1 -10624.415,E2 -10624.415} C_VEL
LIN {X 0,Y 410.941,Z 382.15,A -85,B 0,C 180,E1 -10625.396,E2 -10625.396} C_VEL
LIN {X 0,Y 411.068,Z 376.691,A -85,B 0,C 180,E1 -10626.379,E2 -10626.379} C_VEL
LIN {X 0,Y 411.198,Z 368.896,A -85,B 0,C 180,E1 -10627.453,E2 -10627.453} C_VEL
LIN {X 0,Y 411.472,Z 360.33,A -85,B 0,C 180,E1 -10628.346,E2 -10628.346} C_VEL
LIN {X 0,Y 411.701,Z 350.954,A -85,B 0,C 180,E1 -10629.084,E2 -10629.084} C_VEL
LIN {X 0,Y 411.583,Z 344.682,A -85,B 0,C 180,E1 -10629.458,E2 -10629.458} C_VEL
LIN {X 0,Y 410.718,Z 338.41,A -85,B 0,C 180,E1 -10629.789,E2 -10629.789} C_VEL
LIN {X 0,Y 410.813,Z 331.287,A -85,B 0,C 180,E1 -10632.848,E2 -10632.848} C_VEL
LIN {X 0,Y 410.806,Z 322.556,A -85,B 0,C 180,E1 -10636.656,E2 -10636.656} C_VEL
LIN {X 0,Y 410.927,Z 314.901,A -85,B 0,C 180,E1 -10640.001,E2 -10640.001} C_VEL
LIN {X 0,Y 410.981,Z 306.511,A -85,B 0,C 180,E1 -10643.693,E2 -10643.693} C_VEL
LIN {X 0,Y 411.104,Z 299.371,A -85,B 0,C 180,E1 -10646.822,E2 -10646.822} C_VEL
LIN {X 0,Y 411.249,Z 293.26,A -85,B 0,C 180,E1 -10649.535,E2 -10649.535} C_VEL
LIN {X 0,Y 411.199,Z 293.266,A -85,B 0,C 180,E1 -10653.155,E2 -10653.155} C_VEL
LIN {X 0,Y 411.186,Z 293.264,A -85,B 0,C 180,E1 -10656.551,E2 -10656.551} C_VEL
LIN {X 0,Y 411.171,Z 293.266,A -85,B 0,C 180,E1 -10659.72,E2 -10659.72} C_VEL
LIN {X 0,Y 411.162,Z 293.27,A -85,B 0,C 180,E1 -10663.133,E2 -10663.133} C_VEL
LIN {X 0,Y 411.16,Z 293.268,A -85,B 0,C 180,E1 -10665.88,E2 -10665.88} C_VEL
LIN {X 0,Y 411.157,Z 293.272,A -85,B 0,C 180,E1 -10668.77,E2 -10668.77} C_VEL
LIN {X 0,Y 411.203,Z 293.263,A -85,B 0,C 180,E1 -10671.829,E2 -10671.829} C_VEL
LIN {X 0,Y 411.202,Z 293.264,A -85,B 0,C 180,E1 -10675.12,E2 -10675.12} C_VEL
LIN {X 0,Y 411.162,Z 293.269,A -85,B 0,C 180,E1 -10678.002,E2 -10678.002} C_VEL
LIN {X 0,Y 411.214,Z 293.262,A -85,B 0,C 180,E1 -10681.41,E2 -10681.41} C_VEL
LIN {X 0,Y 411.226,Z 293.262,A -85,B 0,C 180,E1 -10684.706,E2 -10684.706} C_VEL
LIN {X 0,Y 411.194,Z 293.265,A -85,B 0,C 180,E1 -10687.913,E2 -10687.913} C_VEL
LIN {X 0,Y 411.213,Z 293.262,A -85,B 0,C 180,E1 -10691.051,E2 -10691.051} C_VEL
LIN {X 0,Y 411.243,Z 293.259,A -85,B 0,C 180,E1 -10694.131,E2 -10694.131} C_VEL
LIN {X 0,Y 411.291,Z 293.251,A -85,B 0,C 180,E1 -10697.165,E2 -10697.165} C_VEL
LIN {X 0,Y 411.278,Z 293.256,A -85,B 0,C 180,E1 -10700.161,E2 -10700.161} C_VEL
LIN {X 0,Y 411.381,Z 293.239,A -85,B 0,C 180,E1 -10703.132,E2 -10703.132} C_VEL
LIN {X 0,Y 411.284,Z 293.251,A -85,B 0,C 180,E1 -10705.099,E2 -10705.099} C_VEL
LIN {X 0,Y 411.489,Z 293.231,A -85,B 0,C 180,E1 -10708.042,E2 -10708.042} C_VEL
LIN {X 0,Y 411.363,Z 293.24,A -85,B 0,C 180,E1 -10710.979,E2 -10710.979} C_VEL
LIN {X 0,Y 411.419,Z 293.234,A -85,B 0,C 180,E1 -10712.938,E2 -10712.938} C_VEL
LIN {X 0,Y 411.423,Z 293.238,A -85,B 0,C 180,E1 -10715.883,E2 -10715.883} C_VEL
LIN {X 0,Y 411.306,Z 293.249,A -85,B 0,C 180,E1 -10718.846,E2 -10718.846} C_VEL
LIN {X 0,Y 411.27,Z 293.253,A -85,B 0,C 180,E1 -10722.502,E2 -10722.502} C_VEL
LIN {X 0,Y 411.243,Z 293.259,A -85,B 0,C 180,E1 -10725.869,E2 -10725.869} C_VEL
LIN {X 0,Y 411.244,Z 293.257,A -85,B 0,C 180,E1 -10726.748,E2 -10726.748} C_VEL
LIN {X 0,Y 410.604,Z 293.34,A -85,B 0,C 180,E1 -10727.565,E2 -10727.565} C_VEL
LIN {X 0,Y 407.72,Z 293.697,A -85,B 0,C 180,E1 -10728.893,E2 -10728.893} C_VEL
LIN {X 0,Y 405.259,Z 294.004,A -85,B 0,C 180,E1 -10729.965,E2 -10729.965} C_VEL
LIN {X 0,Y 404.204,Z 294.135,A -85,B 0,C 180,E1 -10730.794,E2 -10730.794} C_VEL
LIN {X 0,Y 404.12,Z 294.145,A -85,B 0,C 180,E1 -10731.075,E2 -10731.075} C_VEL
LIN {X 0,Y 404.159,Z 294.142,A -85,B 0,C 180,E1 -10733.575,E2 -10733.575} C_VEL
LIN {X 0,Y 404.173,Z 294.14,A -85,B 0,C 180,E1 -10735.767,E2 -10735.767} C_VEL
LIN {X 0,Y 404.188,Z 294.138,A -85,B 0,C 180,E1 -10738,E2 -10738} C_VEL
LIN {X 0,Y 404.136,Z 294.145,A -85,B 0,C 180,E1 -10741.561,E2 -10741.561} C_VEL
LIN {X 0,Y 404.176,Z 294.139,A -85,B 0,C 180,E1 -10745.017,E2 -10745.017} C_VEL
LIN {X 0,Y 404.151,Z 294.142,A -85,B 0,C 180,E1 -10748.758,E2 -10748.758} C_VEL
LIN {X 0,Y 404.115,Z 294.147,A -85,B 0,C 180,E1 -10751.601,E2 -10751.601} C_VEL
LIN {X 0,Y 404.138,Z 294.143,A -85,B 0,C 180,E1 -10754.523,E2 -10754.523} C_VEL
LIN {X 0,Y 404.124,Z 294.146,A -85,B 0,C 180,E1 -10757.296,E2 -10757.296} C_VEL
LIN {X 0,Y 404.125,Z 294.143,A -85,B 0,C 180,E1 -10759.952,E2 -10759.952} C_VEL
LIN {X 0,Y 404.128,Z 294.145,A -85,B 0,C 180,E1 -10763.127,E2 -10763.127} C_VEL
LIN {X 0,Y 404.133,Z 294.142,A -85,B 0,C 180,E1 -10766.189,E2 -10766.189} C_VEL
LIN {X 0,Y 404.317,Z 294.23,A -85,B 0,C 180,E1 -10769.153,E2 -10769.153} C_VEL
LIN {X 0,Y 404.34,Z 298.412,A -85,B 0,C 180,E1 -10771.448,E2 -10771.448} C_VEL
LIN {X 0,Y 404.013,Z 304.573,A -85,B 0,C 180,E1 -10774.765,E2 -10774.765} C_VEL
LIN {X 0,Y 403.768,Z 311.755,A -85,B 0,C 180,E1 -10778.562,E2 -10778.562} C_VEL
LIN {X 0,Y 403.582,Z 317.857,A -85,B 0,C 180,E1 -10781.734,E2 -10781.734} C_VEL
LIN {X 0,Y 403.384,Z 323.962,A -85,B 0,C 180,E1 -10784.852,E2 -10784.852} C_VEL
LIN {X 0,Y 403.327,Z 330.066,A -85,B 0,C 180,E1 -10787.932,E2 -10787.932} C_VEL
LIN {X 0,Y 403.254,Z 333.325,A -85,B 0,C 180,E1 -10789.457,E2 -10789.457} C_VEL
LIN {X 0,Y 404.757,Z 344.175,A -85,B 0,C 180,E1 -10790.065,E2 -10790.065} C_VEL
LIN {X 0,Y 405.025,Z 350.548,A -85,B 0,C 180,E1 -10790.513,E2 -10790.513} C_VEL
LIN {X 0,Y 404.655,Z 360.581,A -85,B 0,C 180,E1 -10791.386,E2 -10791.386} C_VEL
LIN {X 0,Y 404.307,Z 368.15,A -85,B 0,C 180,E1 -10792.233,E2 -10792.233} C_VEL
LIN {X 0,Y 404.097,Z 375.466,A -85,B 0,C 180,E1 -10793.26,E2 -10793.26} C_VEL
LIN {X 0,Y 403.929,Z 382.404,A -85,B 0,C 180,E1 -10794.51,E2 -10794.51} C_VEL
LIN {X 0,Y 403.715,Z 386.758,A -85,B 0,C 180,E1 -10795.508,E2 -10795.508} C_VEL
LIN {X 0,Y 403.597,Z 390.201,A -85,B 0,C 180,E1 -10796.507,E2 -10796.507} C_VEL
LIN {X 0,Y 403.283,Z 393.901,A -85,B 0,C 180,E1 -10798.004,E2 -10798.004} C_VEL
LIN {X 0,Y 403.202,Z 395.474,A -85,B 0,C 180,E1 -10799.003,E2 -10799.003} C_VEL
LIN {X 0,Y 403.204,Z 396.369,A -85,B 0,C 180,E1 -10800.001,E2 -10800.001} C_VEL
LIN {X 0,Y 403.262,Z 396.594,A -85,B 0,C 180,E1 -10801,E2 -10801} C_VEL
LIN {X 0,Y 403.368,Z 396.153,A -85,B 0,C 180,E1 -10801.998,E2 -10801.998} C_VEL
LIN {X 0,Y 403.548,Z 395.041,A -85,B 0,C 180,E1 -10802.996,E2 -10802.996} C_VEL
LIN {X 0,Y 404.153,Z 392.036,A -85,B 0,C 180,E1 -10804.489,E2 -10804.489} C_VEL
LIN {X 0,Y 404.353,Z 389.142,A -85,B 0,C 180,E1 -10805.487,E2 -10805.487} C_VEL
LIN {X 0,Y 404.873,Z 384.361,A -85,B 0,C 180,E1 -10806.73,E2 -10806.73} C_VEL
LIN {X 0,Y 405.382,Z 378.073,A -85,B 0,C 180,E1 -10807.973,E2 -10807.973} C_VEL
LIN {X 0,Y 405.961,Z 371.638,A -85,B 0,C 180,E1 -10808.965,E2 -10808.965} C_VEL
LIN {X 0,Y 406.656,Z 363.582,A -85,B 0,C 180,E1 -10809.953,E2 -10809.953} C_VEL
LIN {X 0,Y 407.258,Z 354.634,A -85,B 0,C 180,E1 -10810.818,E2 -10810.818} C_VEL
LIN {X 0,Y 407.021,Z 350.205,A -85,B 0,C 180,E1 -10811.202,E2 -10811.202} C_VEL
LIN {X 0,Y 404.878,Z 340.111,A -85,B 0,C 180,E1 -10812.024,E2 -10812.024} C_VEL
LIN {X 0,Y 404.082,Z 336.775,A -85,B 0,C 180,E1 -10812.293,E2 -10812.293} C_VEL
LIN {X 0,Y 404.294,Z 331.811,A -85,B 0,C 180,E1 -10815.116,E2 -10815.116} C_VEL
LIN {X 0,Y 404.628,Z 326.504,A -85,B 0,C 180,E1 -10818.22,E2 -10818.22} C_VEL
LIN {X 0,Y 405.013,Z 321.351,A -85,B 0,C 180,E1 -10821.372,E2 -10821.372} C_VEL
LIN {X 0,Y 405.493,Z 316.415,A -85,B 0,C 180,E1 -10824.581,E2 -10824.581} C_VEL
LIN {X 0,Y 406.144,Z 311.371,A -85,B 0,C 180,E1 -10828.052,E2 -10828.052} C_VEL
LIN {X 0,Y 406.476,Z 308.565,A -85,B 0,C 180,E1 -10830.173,E2 -10830.173} C_VEL
LIN {X 0,Y 406.373,Z 305.935,A -85,B 0,C 180,E1 -10832.422,E2 -10832.422} C_VEL
LIN {X 0,Y 406.151,Z 303.593,A -85,B 0,C 180,E1 -10834.823,E2 -10834.823} C_VEL
LIN {X 0,Y 405.844,Z 301.719,A -85,B 0,C 180,E1 -10837.309,E2 -10837.309} C_VEL
LIN {X 0,Y 405.567,Z 300.244,A -85,B 0,C 180,E1 -10840.317,E2 -10840.317} C_VEL
LIN {X 0,Y 405.504,Z 299.843,A -85,B 0,C 180,E1 -10843.287,E2 -10843.287} C_VEL
LIN {X 0,Y 405.692,Z 300.54,A -85,B 0,C 180,E1 -10846.136,E2 -10846.136} C_VEL
LIN {X 0,Y 406.192,Z 302.355,A -85,B 0,C 180,E1 -10848.892,E2 -10848.892} C_VEL
LIN {X 0,Y 406.916,Z 305.228,A -85,B 0,C 180,E1 -10851.554,E2 -10851.554} C_VEL
LIN {X 0,Y 407.864,Z 309.078,A -85,B 0,C 180,E1 -10854.136,E2 -10854.136} C_VEL
LIN {X 0,Y 408.996,Z 313.795,A -85,B 0,C 180,E1 -10856.642,E2 -10856.642} C_VEL
LIN {X 0,Y 410.066,Z 319.427,A -85,B 0,C 180,E1 -10859.058,E2 -10859.058} C_VEL
LIN {X 0,Y 410.271,Z 322.433,A -85,B 0,C 180,E1 -10860.213,E2 -10860.213} C_VEL
LIN {X 0,Y 408.993,Z 329.14,A -85,B 0,C 180,E1 -10862.357,E2 -10862.357} C_VEL
LIN {X 0,Y 407.193,Z 339.905,A -85,B 0,C 180,E1 -10865.529,E2 -10865.529} C_VEL
LIN {X 0,Y 405.846,Z 351.408,A -85,B 0,C 180,E1 -10868.675,E2 -10868.675} C_VEL
LIN {X 0,Y 404.677,Z 365.668,A -85,B 0,C 180,E1 -10872.333,E2 -10872.333} C_VEL
LIN {X 0,Y 406.628,Z 379.244,A -85,B 0,C 180,E1 -10872.895,E2 -10872.895} C_VEL
LIN {X 0,Y 407.301,Z 391.572,A -85,B 0,C 180,E1 -10873.534,E2 -10873.534} C_VEL
LIN {X 0,Y 406.937,Z 402.198,A -85,B 0,C 180,E1 -10874.216,E2 -10874.216} C_VEL
LIN {X 0,Y 405.945,Z 414.471,A -85,B 0,C 180,E1 -10875.205,E2 -10875.205} C_VEL
LIN {X 0,Y 405.282,Z 424.19,A -85,B 0,C 180,E1 -10876.194,E2 -10876.194} C_VEL
LIN {X 0,Y 404.469,Z 434.235,A -85,B 0,C 180,E1 -10877.455,E2 -10877.455} C_VEL
LIN {X 0,Y 403.858,Z 443.907,A -85,B 0,C 180,E1 -10878.964,E2 -10878.964} C_VEL
LIN {X 0,Y 403.443,Z 451.612,A -85,B 0,C 180,E1 -10880.474,E2 -10880.474} C_VEL
LIN {X 0,Y 403.214,Z 457.811,A -85,B 0,C 180,E1 -10881.985,E2 -10881.985} C_VEL
LIN {X 0,Y 403.121,Z 463.001,A -85,B 0,C 180,E1 -10883.589,E2 -10883.589} C_VEL
LIN {X 0,Y 403.091,Z 466.464,A -85,B 0,C 180,E1 -10884.999,E2 -10884.999} C_VEL
LIN {X 0,Y 403.106,Z 468.346,A -85,B 0,C 180,E1 -10886.001,E2 -10886.001} C_VEL
LIN {X 0,Y 403.206,Z 469.786,A -85,B 0,C 180,E1 -10887.003,E2 -10887.003} C_VEL
LIN {X 0,Y 403.224,Z 470.803,A -85,B 0,C 180,E1 -10888.002,E2 -10888.002} C_VEL
LIN {X 0,Y 403.133,Z 471.354,A -85,B 0,C 180,E1 -10889.001,E2 -10889.001} C_VEL
LIN {X 0,Y 403.115,Z 471.471,A -85,B 0,C 180,E1 -10890,E2 -10890} C_VEL
LIN {X 0,Y 403.131,Z 471.182,A -85,B 0,C 180,E1 -10890.999,E2 -10890.999} C_VEL
LIN {X 0,Y 403.23,Z 470.458,A -85,B 0,C 180,E1 -10891.998,E2 -10891.998} C_VEL
LIN {X 0,Y 403.285,Z 469.265,A -85,B 0,C 180,E1 -10892.997,E2 -10892.997} C_VEL
LIN {X 0,Y 403.12,Z 466.609,A -85,B 0,C 180,E1 -10894.5,E2 -10894.5} C_VEL
LIN {X 0,Y 403.159,Z 462.868,A -85,B 0,C 180,E1 -10896.004,E2 -10896.004} C_VEL
LIN {X 0,Y 403.205,Z 457.906,A -85,B 0,C 180,E1 -10897.512,E2 -10897.512} C_VEL
LIN {X 0,Y 403.344,Z 451.568,A -85,B 0,C 180,E1 -10899.022,E2 -10899.022} C_VEL
LIN {X 0,Y 403.659,Z 443.521,A -85,B 0,C 180,E1 -10900.534,E2 -10900.534} C_VEL
LIN {X 0,Y 404.084,Z 435.259,A -85,B 0,C 180,E1 -10901.792,E2 -10901.792} C_VEL
LIN {X 0,Y 404.742,Z 426.235,A -85,B 0,C 180,E1 -10902.918,E2 -10902.918} C_VEL
LIN {X 0,Y 405.031,Z 417.711,A -85,B 0,C 180,E1 -10903.797,E2 -10903.797} C_VEL
LIN {X 0,Y 405.565,Z 407.218,A -85,B 0,C 180,E1 -10904.681,E2 -10904.681} C_VEL
LIN {X 0,Y 406.202,Z 394.717,A -85,B 0,C 180,E1 -10905.492,E2 -10905.492} C_VEL
LIN {X 0,Y 405.61,Z 382.945,A -85,B 0,C 180,E1 -10906.079,E2 -10906.079} C_VEL
LIN {X 0,Y 404.39,Z 370.017,A -85,B 0,C 180,E1 -10906.53,E2 -10906.53} C_VEL
LIN {X 0,Y 404.21,Z 367.111,A -85,B 0,C 180,E1 -10906.609,E2 -10906.609} C_VEL
LIN {X 0,Y 404.932,Z 354.221,A -85,B 0,C 180,E1 -10909.782,E2 -10909.782} C_VEL
LIN {X 0,Y 406.088,Z 340.552,A -85,B 0,C 180,E1 -10913.187,E2 -10913.187} C_VEL
LIN {X 0,Y 407.582,Z 325.825,A -85,B 0,C 180,E1 -10916.913,E2 -10916.913} C_VEL
LIN {X 0,Y 408.58,Z 316.327,A -85,B 0,C 180,E1 -10919.356,E2 -10919.356} C_VEL
LIN {X 0,Y 407.478,Z 309.866,A -85,B 0,C 180,E1 -10921.16,E2 -10921.16} C_VEL
LIN {X 0,Y 404.988,Z 298.007,A -85,B 0,C 180,E1 -10924.634,E2 -10924.634} C_VEL
LIN {X 0,Y 404.189,Z 294.14,A -85,B 0,C 180,E1 -10925.833,E2 -10925.833} C_VEL
LIN {X 0,Y 404.16,Z 294.143,A -85,B 0,C 180,E1 -10928.757,E2 -10928.757} C_VEL
LIN {X 0,Y 404.128,Z 294.145,A -85,B 0,C 180,E1 -10931.599,E2 -10931.599} C_VEL
LIN {X 0,Y 404.151,Z 294.143,A -85,B 0,C 180,E1 -10934.522,E2 -10934.522} C_VEL
LIN {X 0,Y 404.142,Z 294.145,A -85,B 0,C 180,E1 -10937.295,E2 -10937.295} C_VEL
LIN {X 0,Y 404.174,Z 294.139,A -85,B 0,C 180,E1 -10939.955,E2 -10939.955} C_VEL
LIN {X 0,Y 404.142,Z 294.146,A -85,B 0,C 180,E1 -10943.124,E2 -10943.124} C_VEL
LIN {X 0,Y 404.15,Z 294.147,A -85,B 0,C 180,E1 -10946.187,E2 -10946.187} C_VEL
LIN {X 0,Y 404.163,Z 294.232,A -85,B 0,C 180,E1 -10948.627,E2 -10948.627} C_VEL
LIN {X 0,Y 405.069,Z 299.65,A -85,B 0,C 180,E1 -10950.934,E2 -10950.934} C_VEL
LIN {X 0,Y 404.958,Z 306.453,A -85,B 0,C 180,E1 -10953.732,E2 -10953.732} C_VEL
LIN {X 0,Y 404.779,Z 313.982,A -85,B 0,C 180,E1 -10956.958,E2 -10956.958} C_VEL
LIN {X 0,Y 404.71,Z 320.429,A -85,B 0,C 180,E1 -10959.676,E2 -10959.676} C_VEL
LIN {X 0,Y 404.526,Z 328.901,A -85,B 0,C 180,E1 -10963.352,E2 -10963.352} C_VEL
LIN {X 0,Y 404.473,Z 337.018,A -85,B 0,C 180,E1 -10966.944,E2 -10966.944} C_VEL
LIN {X 0,Y 404.386,Z 341.889,A -85,B 0,C 180,E1 -10969.104,E2 -10969.104} C_VEL
LIN {X 0,Y 406.179,Z 350.366,A -85,B 0,C 180,E1 -10969.657,E2 -10969.657} C_VEL
LIN {X 0,Y 405.923,Z 359.247,A -85,B 0,C 180,E1 -10970.305,E2 -10970.305} C_VEL
LIN {X 0,Y 405.525,Z 367.634,A -85,B 0,C 180,E1 -10971.128,E2 -10971.128} C_VEL
LIN {X 0,Y 405.059,Z 374.728,A -85,B 0,C 180,E1 -10972.02,E2 -10972.02} C_VEL
LIN {X 0,Y 404.777,Z 380.79,A -85,B 0,C 180,E1 -10973.018,E2 -10973.018} C_VEL
LIN {X 0,Y 404.37,Z 386.68,A -85,B 0,C 180,E1 -10974.263,E2 -10974.263} C_VEL
LIN {X 0,Y 404.141,Z 390.873,A -85,B 0,C 180,E1 -10975.51,E2 -10975.51} C_VEL
LIN {X 0,Y 403.848,Z 392.267,A -85,B 0,C 180,E1 -10976.007,E2 -10976.007} C_VEL
LIN {X 0,Y 403.512,Z 394.317,A -85,B 0,C 180,E1 -10977.004,E2 -10977.004} C_VEL
LIN {X 0,Y 403.332,Z 395.615,A -85,B 0,C 180,E1 -10978.002,E2 -10978.002} C_VEL
LIN {X 0,Y 403.232,Z 396.216,A -85,B 0,C 180,E1 -10979,E2 -10979} C_VEL
LIN {X 0,Y 403.183,Z 396.132,A -85,B 0,C 180,E1 -10979.999,E2 -10979.999} C_VEL
LIN {X 0,Y 403.189,Z 395.361,A -85,B 0,C 180,E1 -10980.997,E2 -10980.997} C_VEL
LIN {X 0,Y 403.343,Z 392.902,A -85,B 0,C 180,E1 -10982.495,E2 -10982.495} C_VEL
LIN {X 0,Y 403.587,Z 388.703,A -85,B 0,C 180,E1 -10983.993,E2 -10983.993} C_VEL
LIN {X 0,Y 403.875,Z 383.6,A -85,B 0,C 180,E1 -10985.24,E2 -10985.24} C_VEL
LIN {X 0,Y 403.97,Z 378.351,A -85,B 0,C 180,E1 -10986.241,E2 -10986.241} C_VEL
LIN {X 0,Y 404.09,Z 371.54,A -85,B 0,C 180,E1 -10987.248,E2 -10987.248} C_VEL
LIN {X 0,Y 404.324,Z 364.076,A -85,B 0,C 180,E1 -10988.118,E2 -10988.118} C_VEL
LIN {X 0,Y 404.516,Z 355.646,A -85,B 0,C 180,E1 -10988.869,E2 -10988.869} C_VEL
LIN {X 0,Y 404.665,Z 346.301,A -85,B 0,C 180,E1 -10989.495,E2 -10989.495} C_VEL
LIN {X 0,Y 403.664,Z 338.953,A -85,B 0,C 180,E1 -10989.899,E2 -10989.899} C_VEL
LIN {X 0,Y 403.75,Z 331.575,A -85,B 0,C 180,E1 -10993.077,E2 -10993.077} C_VEL
LIN {X 0,Y 403.753,Z 323.073,A -85,B 0,C 180,E1 -10996.79,E2 -10996.79} C_VEL
LIN {X 0,Y 403.876,Z 315.755,A -85,B 0,C 180,E1 -11000.002,E2 -11000.002} C_VEL
LIN {X 0,Y 403.946,Z 307.639,A -85,B 0,C 180,E1 -11003.587,E2 -11003.587} C_VEL
LIN {X 0,Y 404.048,Z 300.051,A -85,B 0,C 180,E1 -11006.886,E2 -11006.886} C_VEL
LIN {X 0,Y 404.216,Z 294.136,A -85,B 0,C 180,E1 -11009.52,E2 -11009.52} C_VEL
LIN {X 0,Y 404.162,Z 294.142,A -85,B 0,C 180,E1 -11013.418,E2 -11013.418} C_VEL
LIN {X 0,Y 404.134,Z 294.141,A -85,B 0,C 180,E1 -11016.245,E2 -11016.245} C_VEL
LIN {X 0,Y 404.131,Z 294.145,A -85,B 0,C 180,E1 -11018.758,E2 -11018.758} C_VEL
LIN {X 0,Y 404.107,Z 294.146,A -85,B 0,C 180,E1 -11021.597,E2 -11021.597} C_VEL
LIN {X 0,Y 404.137,Z 294.144,A -85,B 0,C 180,E1 -11024.521,E2 -11024.521} C_VEL
LIN {X 0,Y 404.128,Z 294.145,A -85,B 0,C 180,E1 -11027.294,E2 -11027.294} C_VEL
LIN {X 0,Y 404.16,Z 294.14,A -85,B 0,C 180,E1 -11029.954,E2 -11029.954} C_VEL
LIN {X 0,Y 404.131,Z 294.145,A -85,B 0,C 180,E1 -11033.123,E2 -11033.123} C_VEL
LIN {X 0,Y 404.136,Z 294.145,A -85,B 0,C 180,E1 -11036.187,E2 -11036.187} C_VEL
LIN {X 0,Y 404.145,Z 294.142,A -85,B 0,C 180,E1 -11039.715,E2 -11039.715} C_VEL
LIN {X 0,Y 404.185,Z 294.139,A -85,B 0,C 180,E1 -11043.122,E2 -11043.122} C_VEL
LIN {X 0,Y 404.166,Z 294.14,A -85,B 0,C 180,E1 -11045.334,E2 -11045.334} C_VEL
LIN {X 0,Y 404.128,Z 294.146,A -85,B 0,C 180,E1 -11048.58,E2 -11048.58} C_VEL
LIN {X 0,Y 404.199,Z 294.136,A -85,B 0,C 180,E1 -11051.761,E2 -11051.761} C_VEL
LIN {X 0,Y 404.194,Z 294.137,A -85,B 0,C 180,E1 -11054.881,E2 -11054.881} C_VEL
LIN {X 0,Y 404.243,Z 294.13,A -85,B 0,C 180,E1 -11057.958,E2 -11057.958} C_VEL
LIN {X 0,Y 404.253,Z 294.128,A -85,B 0,C 180,E1 -11060.998,E2 -11060.998} C_VEL
LIN {X 0,Y 404.37,Z 294.116,A -85,B 0,C 180,E1 -11064.014,E2 -11064.014} C_VEL
LIN {X 0,Y 404.458,Z 294.107,A -85,B 0,C 180,E1 -11068.008,E2 -11068.008} C_VEL
LIN {X 0,Y 404.334,Z 294.116,A -85,B 0,C 180,E1 -11070.996,E2 -11070.996} C_VEL
LIN {X 0,Y 404.379,Z 294.111,A -85,B 0,C 180,E1 -11072.989,E2 -11072.989} C_VEL
LIN {X 0,Y 404.37,Z 294.116,A -85,B 0,C 180,E1 -11075.986,E2 -11075.986} C_VEL
LIN {X 0,Y 404.253,Z 294.128,A -85,B 0,C 180,E1 -11079.002,E2 -11079.002} C_VEL
LIN {X 0,Y 404.243,Z 294.13,A -85,B 0,C 180,E1 -11082.042,E2 -11082.042} C_VEL
LIN {X 0,Y 404.194,Z 294.137,A -85,B 0,C 180,E1 -11085.119,E2 -11085.119} C_VEL
LIN {X 0,Y 404.199,Z 294.136,A -85,B 0,C 180,E1 -11088.239,E2 -11088.239} C_VEL
LIN {X 0,Y 404.12,Z 294.145,A -85,B 0,C 180,E1 -11091.075,E2 -11091.075} C_VEL
LIN {X 0,Y 403.464,Z 294.229,A -85,B 0,C 180,E1 -11091.908,E2 -11091.908} C_VEL
LIN {X 0,Y 400.633,Z 294.584,A -85,B 0,C 180,E1 -11093.261,E2 -11093.261} C_VEL
LIN {X 0,Y 398.239,Z 294.881,A -85,B 0,C 180,E1 -11094.354,E2 -11094.354} C_VEL
LIN {X 0,Y 397.22,Z 295.007,A -85,B 0,C 180,E1 -11095.199,E2 -11095.199} C_VEL
LIN {X 0,Y 397.142,Z 295.016,A -85,B 0,C 180,E1 -11095.485,E2 -11095.485} C_VEL
LIN {X 0,Y 397.117,Z 295.018,A -85,B 0,C 180,E1 -11098.544,E2 -11098.544} C_VEL
LIN {X 0,Y 397.073,Z 295.023,A -85,B 0,C 180,E1 -11102.072,E2 -11102.072} C_VEL
LIN {X 0,Y 397.111,Z 295.021,A -85,B 0,C 180,E1 -11105.505,E2 -11105.505} C_VEL
LIN {X 0,Y 397.125,Z 295.017,A -85,B 0,C 180,E1 -11108.863,E2 -11108.863} C_VEL
LIN {X 0,Y 397.061,Z 295.024,A -85,B 0,C 180,E1 -11112.268,E2 -11112.268} C_VEL
LIN {X 0,Y 397.079,Z 295.025,A -85,B 0,C 180,E1 -11115.07,E2 -11115.07} C_VEL
LIN {X 0,Y 397.051,Z 295.024,A -85,B 0,C 180,E1 -11118.024,E2 -11118.024} C_VEL
LIN {X 0,Y 397.085,Z 295.02,A -85,B 0,C 180,E1 -11121.725,E2 -11121.725} C_VEL
LIN {X 0,Y 397.114,Z 295.016,A -85,B 0,C 180,E1 -11125.508,E2 -11125.508} C_VEL
LIN {X 0,Y 397.286,Z 295.181,A -85,B 0,C 180,E1 -11129.137,E2 -11129.137} C_VEL
LIN {X 0,Y 397.304,Z 299.379,A -85,B 0,C 180,E1 -11131.472,E2 -11131.472} C_VEL
LIN {X 0,Y 396.966,Z 305.607,A -85,B 0,C 180,E1 -11134.857,E2 -11134.857} C_VEL
LIN {X 0,Y 396.733,Z 311.793,A -85,B 0,C 180,E1 -11138.162,E2 -11138.162} C_VEL
LIN {X 0,Y 396.562,Z 317.942,A -85,B 0,C 180,E1 -11141.399,E2 -11141.399} C_VEL
LIN {X 0,Y 396.345,Z 324.094,A -85,B 0,C 180,E1 -11144.576,E2 -11144.576} C_VEL
LIN {X 0,Y 396.281,Z 330.25,A -85,B 0,C 180,E1 -11147.714,E2 -11147.714} C_VEL
LIN {X 0,Y 396.163,Z 333.41,A -85,B 0,C 180,E1 -11149.298,E2 -11149.298} C_VEL
LIN {X 0,Y 397.723,Z 344.823,A -85,B 0,C 180,E1 -11149.952,E2 -11149.952} C_VEL
LIN {X 0,Y 398.01,Z 350.312,A -85,B 0,C 180,E1 -11150.344,E2 -11150.344} C_VEL
LIN {X 0,Y 397.639,Z 360.472,A -85,B 0,C 180,E1 -11151.233,E2 -11151.233} C_VEL
LIN {X 0,Y 397.234,Z 369.905,A -85,B 0,C 180,E1 -11152.317,E2 -11152.317} C_VEL
LIN {X 0,Y 397.009,Z 377.168,A -85,B 0,C 180,E1 -11153.394,E2 -11153.394} C_VEL
LIN {X 0,Y 396.837,Z 383.862,A -85,B 0,C 180,E1 -11154.666,E2 -11154.666} C_VEL
LIN {X 0,Y 396.553,Z 388.963,A -85,B 0,C 180,E1 -11155.936,E2 -11155.936} C_VEL
LIN {X 0,Y 396.348,Z 392.088,A -85,B 0,C 180,E1 -11156.952,E2 -11156.952} C_VEL
LIN {X 0,Y 396.234,Z 394.44,A -85,B 0,C 180,E1 -11157.968,E2 -11157.968} C_VEL
LIN {X 0,Y 396.145,Z 396.084,A -85,B 0,C 180,E1 -11158.985,E2 -11158.985} C_VEL
LIN {X 0,Y 396.143,Z 397.045,A -85,B 0,C 180,E1 -11160.001,E2 -11160.001} C_VEL
LIN {X 0,Y 396.203,Z 397.333,A -85,B 0,C 180,E1 -11161.018,E2 -11161.018} C_VEL
LIN {X 0,Y 396.319,Z 396.954,A -85,B 0,C 180,E1 -11162.034,E2 -11162.034} C_VEL
LIN {X 0,Y 396.513,Z 395.916,A -85,B 0,C 180,E1 -11163.049,E2 -11163.049} C_VEL
LIN {X 0,Y 397.142,Z 393.047,A -85,B 0,C 180,E1 -11164.569,E2 -11164.569} C_VEL
LIN {X 0,Y 397.391,Z 390.259,A -85,B 0,C 180,E1 -11165.583,E2 -11165.583} C_VEL
LIN {X 0,Y 397.938,Z 385.588,A -85,B 0,C 180,E1 -11166.848,E2 -11166.848} C_VEL
LIN {X 0,Y 398.474,Z 379.459,A -85,B 0,C 180,E1 -11168.113,E2 -11168.113} C_VEL
LIN {X 0,Y 399.214,Z 371.866,A -85,B 0,C 180,E1 -11169.312,E2 -11169.312} C_VEL
LIN {X 0,Y 399.979,Z 363.465,A -85,B 0,C 180,E1 -11170.351,E2 -11170.351} C_VEL
LIN {X 0,Y 400.622,Z 354.157,A -85,B 0,C 180,E1 -11171.255,E2 -11171.255} C_VEL
LIN {X 0,Y 399.034,Z 345.012,A -85,B 0,C 180,E1 -11172.074,E2 -11172.074} C_VEL
LIN {X 0,Y 397.146,Z 337.313,A -85,B 0,C 180,E1 -11172.684,E2 -11172.684} C_VEL
LIN {X 0,Y 397.446,Z 330.893,A -85,B 0,C 180,E1 -11176.436,E2 -11176.436} C_VEL
LIN {X 0,Y 397.81,Z 325.68,A -85,B 0,C 180,E1 -11179.614,E2 -11179.614} C_VEL
LIN {X 0,Y 398.298,Z 320.643,A -85,B 0,C 180,E1 -11182.843,E2 -11182.843} C_VEL
LIN {X 0,Y 398.861,Z 315.871,A -85,B 0,C 180,E1 -11186.137,E2 -11186.137} C_VEL
LIN {X 0,Y 399.338,Z 312.764,A -85,B 0,C 180,E1 -11188.372,E2 -11188.372} C_VEL
LIN {X 0,Y 399.612,Z 309.898,A -85,B 0,C 180,E1 -11190.667,E2 -11190.667} C_VEL
LIN {X 0,Y 399.533,Z 307.372,A -85,B 0,C 180,E1 -11193.047,E2 -11193.047} C_VEL
LIN {X 0,Y 399.262,Z 304.893,A -85,B 0,C 180,E1 -11195.932,E2 -11195.932} C_VEL
LIN {X 0,Y 398.93,Z 303.042,A -85,B 0,C 180,E1 -11199.181,E2 -11199.181} C_VEL
LIN {X 0,Y 398.825,Z 302.356,A -85,B 0,C 180,E1 -11202.039,E2 -11202.039} C_VEL
LIN {X 0,Y 398.912,Z 302.627,A -85,B 0,C 180,E1 -11204.808,E2 -11204.808} C_VEL
LIN {X 0,Y 399.33,Z 303.991,A -85,B 0,C 180,E1 -11207.663,E2 -11207.663} C_VEL
LIN {X 0,Y 400.052,Z 306.661,A -85,B 0,C 180,E1 -11210.624,E2 -11210.624} C_VEL
LIN {X 0,Y 400.931,Z 310.402,A -85,B 0,C 180,E1 -11213.416,E2 -11213.416} C_VEL
LIN {X 0,Y 401.707,Z 313.668,A -85,B 0,C 180,E1 -11215.315,E2 -11215.315} C_VEL
LIN {X 0,Y 402.824,Z 318.798,A -85,B 0,C 180,E1 -11217.851,E2 -11217.851} C_VEL
LIN {X 0,Y 403.504,Z 323.22,A -85,B 0,C 180,E1 -11219.662,E2 -11219.662} C_VEL
LIN {X 0,Y 403.138,Z 326.334,A -85,B 0,C 180,E1 -11220.782,E2 -11220.782} C_VEL
LIN {X 0,Y 401.065,Z 336.641,A -85,B 0,C 180,E1 -11224.018,E2 -11224.018} C_VEL
LIN {X 0,Y 399.263,Z 349.621,A -85,B 0,C 180,E1 -11227.762,E2 -11227.762} C_VEL
LIN {X 0,Y 397.86,Z 363.516,A -85,B 0,C 180,E1 -11231.46,E2 -11231.46} C_VEL
LIN {X 0,Y 397.738,Z 365.438,A -85,B 0,C 180,E1 -11231.934,E2 -11231.934} C_VEL
LIN {X 0,Y 399.769,Z 378.429,A -85,B 0,C 180,E1 -11232.502,E2 -11232.502} C_VEL
LIN {X 0,Y 400.411,Z 389.572,A -85,B 0,C 180,E1 -11233.089,E2 -11233.089} C_VEL
LIN {X 0,Y 400.37,Z 398.912,A -85,B 0,C 180,E1 -11233.688,E2 -11233.688} C_VEL
LIN {X 0,Y 399.465,Z 410.37,A -85,B 0,C 180,E1 -11234.567,E2 -11234.567} C_VEL
LIN {X 0,Y 398.496,Z 421.904,A -85,B 0,C 180,E1 -11235.705,E2 -11235.705} C_VEL
LIN {X 0,Y 397.732,Z 432.204,A -85,B 0,C 180,E1 -11236.98,E2 -11236.98} C_VEL
LIN {X 0,Y 397.083,Z 440.592,A -85,B 0,C 180,E1 -11238.256,E2 -11238.256} C_VEL
LIN {X 0,Y 396.447,Z 448.825,A -85,B 0,C 180,E1 -11239.789,E2 -11239.789} C_VEL
LIN {X 0,Y 396.204,Z 455.447,A -85,B 0,C 180,E1 -11241.328,E2 -11241.328} C_VEL
LIN {X 0,Y 396.096,Z 460.696,A -85,B 0,C 180,E1 -11242.865,E2 -11242.865} C_VEL
LIN {X 0,Y 396.013,Z 464.757,A -85,B 0,C 180,E1 -11244.399,E2 -11244.399} C_VEL
LIN {X 0,Y 396.015,Z 467.734,A -85,B 0,C 180,E1 -11245.929,E2 -11245.929} C_VEL
LIN {X 0,Y 396.133,Z 469.158,A -85,B 0,C 180,E1 -11246.949,E2 -11246.949} C_VEL
LIN {X 0,Y 396.173,Z 470.156,A -85,B 0,C 180,E1 -11247.967,E2 -11247.967} C_VEL
LIN {X 0,Y 396.08,Z 470.666,A -85,B 0,C 180,E1 -11248.983,E2 -11248.983} C_VEL
LIN {X 0,Y 396.059,Z 470.764,A -85,B 0,C 180,E1 -11250,E2 -11250} C_VEL
LIN {X 0,Y 396.079,Z 470.454,A -85,B 0,C 180,E1 -11251.017,E2 -11251.017} C_VEL
LIN {X 0,Y 396.182,Z 469.683,A -85,B 0,C 180,E1 -11252.033,E2 -11252.033} C_VEL
LIN {X 0,Y 396.208,Z 468.463,A -85,B 0,C 180,E1 -11253.05,E2 -11253.05} C_VEL
LIN {X 0,Y 396.042,Z 465.752,A -85,B 0,C 180,E1 -11254.58,E2 -11254.58} C_VEL
LIN {X 0,Y 396.1,Z 461.951,A -85,B 0,C 180,E1 -11256.111,E2 -11256.111} C_VEL
LIN {X 0,Y 396.149,Z 456.917,A -85,B 0,C 180,E1 -11257.646,E2 -11257.646} C_VEL
LIN {X 0,Y 396.299,Z 450.45,A -85,B 0,C 180,E1 -11259.184,E2 -11259.184} C_VEL
LIN {X 0,Y 396.635,Z 442.295,A -85,B 0,C 180,E1 -11260.722,E2 -11260.722} C_VEL
LIN {X 0,Y 397.017,Z 433.894,A -85,B 0,C 180,E1 -11262.005,E2 -11262.005} C_VEL
LIN {X 0,Y 397.666,Z 424.642,A -85,B 0,C 180,E1 -11263.152,E2 -11263.152} C_VEL
LIN {X 0,Y 398.104,Z 415.466,A -85,B 0,C 180,E1 -11264.087,E2 -11264.087} C_VEL
LIN {X 0,Y 398.714,Z 403.382,A -85,B 0,C 180,E1 -11265.07,E2 -11265.07} C_VEL
LIN {X 0,Y 399.19,Z 393.294,A -85,B 0,C 180,E1 -11265.705,E2 -11265.705} C_VEL
LIN {X 0,Y 398.332,Z 380.863,A -85,B 0,C 180,E1 -11266.315,E2 -11266.315} C_VEL
LIN {X 0,Y 397.292,Z 368.633,A -85,B 0,C 180,E1 -11266.73,E2 -11266.73} C_VEL
LIN {X 0,Y 397.145,Z 366.846,A -85,B 0,C 180,E1 -11266.784,E2 -11266.784} C_VEL
LIN {X 0,Y 397.883,Z 354.565,A -85,B 0,C 180,E1 -11269.878,E2 -11269.878} C_VEL
LIN {X 0,Y 398.907,Z 343.061,A -85,B 0,C 180,E1 -11272.805,E2 -11272.805} C_VEL
LIN {X 0,Y 400.469,Z 327.869,A -85,B 0,C 180,E1 -11276.727,E2 -11276.727} C_VEL
LIN {X 0,Y 401.598,Z 317.917,A -85,B 0,C 180,E1 -11279.341,E2 -11279.341} C_VEL
LIN {X 0,Y 400.884,Z 312.792,A -85,B 0,C 180,E1 -11280.791,E2 -11280.791} C_VEL
LIN {X 0,Y 398.304,Z 300.711,A -85,B 0,C 180,E1 -11284.377,E2 -11284.377} C_VEL
LIN {X 0,Y 397.117,Z 295.02,A -85,B 0,C 180,E1 -11286.204,E2 -11286.204} C_VEL
LIN {X 0,Y 397.119,Z 295.018,A -85,B 0,C 180,E1 -11289.577,E2 -11289.577} C_VEL
LIN {X 0,Y 397.108,Z 295.019,A -85,B 0,C 180,E1 -11293.479,E2 -11293.479} C_VEL
LIN {X 0,Y 397.108,Z 295.018,A -85,B 0,C 180,E1 -11296.52,E2 -11296.52} C_VEL
LIN {X 0,Y 397.12,Z 295.021,A -85,B 0,C 180,E1 -11300.422,E2 -11300.422} C_VEL
LIN {X 0,Y 397.113,Z 295.022,A -85,B 0,C 180,E1 -11304.265,E2 -11304.265} C_VEL
LIN {X 0,Y 397.119,Z 295.025,A -85,B 0,C 180,E1 -11306.726,E2 -11306.726} C_VEL
LIN {X 0,Y 397.119,Z 295.116,A -85,B 0,C 180,E1 -11308.094,E2 -11308.094} C_VEL
LIN {X 0,Y 398.114,Z 300.342,A -85,B 0,C 180,E1 -11310.376,E2 -11310.376} C_VEL
LIN {X 0,Y 398.24,Z 304.03,A -85,B 0,C 180,E1 -11311.932,E2 -11311.932} C_VEL
LIN {X 0,Y 397.941,Z 312.366,A -85,B 0,C 180,E1 -11315.478,E2 -11315.478} C_VEL
LIN {X 0,Y 397.814,Z 318.689,A -85,B 0,C 180,E1 -11318.222,E2 -11318.222} C_VEL
LIN {X 0,Y 397.683,Z 326.181,A -85,B 0,C 180,E1 -11321.451,E2 -11321.451} C_VEL
LIN {X 0,Y 397.535,Z 333.315,A -85,B 0,C 180,E1 -11324.621,E2 -11324.621} C_VEL
LIN {X 0,Y 397.497,Z 340.312,A -85,B 0,C 180,E1 -11327.749,E2 -11327.749} C_VEL
LIN {X 0,Y 397.465,Z 342.933,A -85,B 0,C 180,E1 -11328.832,E2 -11328.832} C_VEL
LIN {X 0,Y 399.257,Z 350.762,A -85,B 0,C 180,E1 -11329.348,E2 -11329.348} C_VEL
LIN {X 0,Y 399.229,Z 357.784,A -85,B 0,C 180,E1 -11329.86,E2 -11329.86} C_VEL
LIN {X 0,Y 398.875,Z 366.323,A -85,B 0,C 180,E1 -11330.645,E2 -11330.645} C_VEL
LIN {X 0,Y 398.243,Z 374.07,A -85,B 0,C 180,E1 -11331.587,E2 -11331.587} C_VEL
LIN {X 0,Y 397.947,Z 380.741,A -85,B 0,C 180,E1 -11332.642,E2 -11332.642} C_VEL
LIN {X 0,Y 397.466,Z 386.759,A -85,B 0,C 180,E1 -11333.909,E2 -11333.909} C_VEL
LIN {X 0,Y 397.159,Z 390.44,A -85,B 0,C 180,E1 -11334.923,E2 -11334.923} C_VEL
LIN {X 0,Y 396.828,Z 393.201,A -85,B 0,C 180,E1 -11335.936,E2 -11335.936} C_VEL
LIN {X 0,Y 396.475,Z 395.167,A -85,B 0,C 180,E1 -11336.95,E2 -11336.95} C_VEL
LIN {X 0,Y 396.282,Z 396.4,A -85,B 0,C 180,E1 -11337.966,E2 -11337.966} C_VEL
LIN {X 0,Y 396.174,Z 396.943,A -85,B 0,C 180,E1 -11338.982,E2 -11338.982} C_VEL
LIN {X 0,Y 396.123,Z 396.798,A -85,B 0,C 180,E1 -11339.999,E2 -11339.999} C_VEL
LIN {X 0,Y 396.133,Z 395.962,A -85,B 0,C 180,E1 -11341.015,E2 -11341.015} C_VEL
LIN {X 0,Y 396.292,Z 393.379,A -85,B 0,C 180,E1 -11342.54,E2 -11342.54} C_VEL
LIN {X 0,Y 396.523,Z 390.677,A -85,B 0,C 180,E1 -11343.555,E2 -11343.555} C_VEL
LIN {X 0,Y 396.731,Z 386.147,A -85,B 0,C 180,E1 -11344.826,E2 -11344.826} C_VEL
LIN {X 0,Y 396.84,Z 381.304,A -85,B 0,C 180,E1 -11345.843,E2 -11345.843} C_VEL
LIN {X 0,Y 396.99,Z 375.191,A -85,B 0,C 180,E1 -11346.862,E2 -11346.862} C_VEL
LIN {X 0,Y 397.146,Z 367.207,A -85,B 0,C 180,E1 -11347.894,E2 -11347.894} C_VEL
LIN {X 0,Y 397.428,Z 358.314,A -85,B 0,C 180,E1 -11348.772,E2 -11348.772} C_VEL
LIN {X 0,Y 397.684,Z 348.502,A -85,B 0,C 180,E1 -11349.471,E2 -11349.471} C_VEL
LIN {X 0,Y 396.615,Z 339.63,A -85,B 0,C 180,E1 -11349.947,E2 -11349.947} C_VEL
LIN {X 0,Y 396.699,Z 331.838,A -85,B 0,C 180,E1 -11353.314,E2 -11353.314} C_VEL
LIN {X 0,Y 396.712,Z 323.576,A -85,B 0,C 180,E1 -11356.932,E2 -11356.932} C_VEL
LIN {X 0,Y 396.836,Z 316.228,A -85,B 0,C 180,E1 -11360.176,E2 -11360.176} C_VEL
LIN {X 0,Y 396.923,Z 307.517,A -85,B 0,C 180,E1 -11364.03,E2 -11364.03} C_VEL
LIN {X 0,Y 397.026,Z 299.862,A -85,B 0,C 180,E1 -11367.401,E2 -11367.401} C_VEL
LIN {X 0,Y 397.189,Z 295.01,A -85,B 0,C 180,E1 -11369.624,E2 -11369.624} C_VEL
LIN {X 0,Y 397.092,Z 295.02,A -85,B 0,C 180,E1 -11373.712,E2 -11373.712} C_VEL
LIN {X 0,Y 397.091,Z 295.023,A -85,B 0,C 180,E1 -11376.994,E2 -11376.994} C_VEL
LIN {X 0,Y 397.05,Z 295.025,A -85,B 0,C 180,E1 -11380.436,E2 -11380.436} C_VEL
LIN {X 0,Y 397.092,Z 295.02,A -85,B 0,C 180,E1 -11383.647,E2 -11383.647} C_VEL
LIN {X 0,Y 397.094,Z 295.022,A -85,B 0,C 180,E1 -11386.52,E2 -11386.52} C_VEL
LIN {X 0,Y 397.107,Z 295.02,A -85,B 0,C 180,E1 -11390.422,E2 -11390.422} C_VEL
LIN {X 0,Y 397.1,Z 295.021,A -85,B 0,C 180,E1 -11394.264,E2 -11394.264} C_VEL
LIN {X 0,Y 397.106,Z 295.021,A -85,B 0,C 180,E1 -11396.726,E2 -11396.726} C_VEL
LIN {X 0,Y 397.124,Z 295.019,A -85,B 0,C 180,E1 -11400.296,E2 -11400.296} C_VEL
LIN {X 0,Y 397.184,Z 295.011,A -85,B 0,C 180,E1 -11402.609,E2 -11402.609} C_VEL
LIN {X 0,Y 397.122,Z 295.018,A -85,B 0,C 180,E1 -11405.981,E2 -11405.981} C_VEL
LIN {X 0,Y 397.127,Z 295.016,A -85,B 0,C 180,E1 -11409.704,E2 -11409.704} C_VEL
LIN {X 0,Y 397.17,Z 295.012,A -85,B 0,C 180,E1 -11412.844,E2 -11412.844} C_VEL
LIN {X 0,Y 397.217,Z 295.007,A -85,B 0,C 180,E1 -11416.702,E2 -11416.702} C_VEL
LIN {X 0,Y 397.204,Z 295.007,A -85,B 0,C 180,E1 -11419.809,E2 -11419.809} C_VEL
LIN {X 0,Y 397.283,Z 294.996,A -85,B 0,C 180,E1 -11422.887,E2 -11422.887} C_VEL
LIN {X 0,Y 397.226,Z 295.002,A -85,B 0,C 180,E1 -11424.925,E2 -11424.925} C_VEL
LIN {X 0,Y 397.427,Z 294.982,A -85,B 0,C 180,E1 -11427.973,E2 -11427.973} C_VEL
LIN {X 0,Y 397.305,Z 294.992,A -85,B 0,C 180,E1 -11431.014,E2 -11431.014} C_VEL
LIN {X 0,Y 397.314,Z 294.991,A -85,B 0,C 180,E1 -11433.042,E2 -11433.042} C_VEL
LIN {X 0,Y 397.321,Z 294.993,A -85,B 0,C 180,E1 -11436.092,E2 -11436.092} C_VEL
LIN {X 0,Y 397.223,Z 295.004,A -85,B 0,C 180,E1 -11439.163,E2 -11439.163} C_VEL
LIN {X 0,Y 397.207,Z 295.007,A -85,B 0,C 180,E1 -11442.259,E2 -11442.259} C_VEL
LIN {X 0,Y 397.167,Z 295.014,A -85,B 0,C 180,E1 -11445.393,E2 -11445.393} C_VEL
LIN {X 0,Y 397.151,Z 295.013,A -85,B 0,C 180,E1 -11448.574,E2 -11448.574} C_VEL
LIN {X 0,Y 397.086,Z 295.023,A -85,B 0,C 180,E1 -11451.819,E2 -11451.819} C_VEL
LIN {X 0,Y 397.146,Z 295.017,A -85,B 0,C 180,E1 -11455.132,E2 -11455.132} C_VEL
LIN {X 0,Y 397.142,Z 295.016,A -85,B 0,C 180,E1 -11455.485,E2 -11455.485} C_VEL
LIN {X 0,Y 396.476,Z 295.099,A -85,B 0,C 180,E1 -11456.332,E2 -11456.332} C_VEL
LIN {X 0,Y 393.586,Z 295.46,A -85,B 0,C 180,E1 -11457.706,E2 -11457.706} C_VEL
LIN {X 0,Y 391.144,Z 295.763,A -85,B 0,C 180,E1 -11458.817,E2 -11458.817} C_VEL
LIN {X 0,Y 390.111,Z 295.893,A -85,B 0,C 180,E1 -11459.677,E2 -11459.677} C_VEL
LIN {X 0,Y 390.036,Z 295.899,A -85,B 0,C 180,E1 -11459.968,E2 -11459.968} C_VEL
LIN {X 0,Y 390.035,Z 295.901,A -85,B 0,C 180,E1 -11462.722,E2 -11462.722} C_VEL
LIN {X 0,Y 390.048,Z 295.898,A -85,B 0,C 180,E1 -11465.827,E2 -11465.827} C_VEL
LIN {X 0,Y 390.064,Z 295.899,A -85,B 0,C 180,E1 -11469.22,E2 -11469.22} C_VEL
LIN {X 0,Y 390.034,Z 295.899,A -85,B 0,C 180,E1 -11472.375,E2 -11472.375} C_VEL
LIN {X 0,Y 390.037,Z 295.901,A -85,B 0,C 180,E1 -11475.356,E2 -11475.356} C_VEL
LIN {X 0,Y 390.013,Z 295.901,A -85,B 0,C 180,E1 -11478.187,E2 -11478.187} C_VEL
LIN {X 0,Y 390.051,Z 295.901,A -85,B 0,C 180,E1 -11480.905,E2 -11480.905} C_VEL
LIN {X 0,Y 390.076,Z 295.899,A -85,B 0,C 180,E1 -11484.794,E2 -11484.794} C_VEL
LIN {X 0,Y 390.236,Z 296.011,A -85,B 0,C 180,E1 -11489.045,E2 -11489.045} C_VEL
LIN {X 0,Y 390.316,Z 299.307,A -85,B 0,C 180,E1 -11490.913,E2 -11490.913} C_VEL
LIN {X 0,Y 389.941,Z 305.583,A -85,B 0,C 180,E1 -11494.372,E2 -11494.372} C_VEL
LIN {X 0,Y 389.707,Z 311.826,A -85,B 0,C 180,E1 -11497.748,E2 -11497.748} C_VEL
LIN {X 0,Y 389.507,Z 318.017,A -85,B 0,C 180,E1 -11501.049,E2 -11501.049} C_VEL
LIN {X 0,Y 389.314,Z 324.206,A -85,B 0,C 180,E1 -11504.291,E2 -11504.291} C_VEL
LIN {X 0,Y 389.183,Z 331.438,A -85,B 0,C 180,E1 -11508.016,E2 -11508.016} C_VEL
LIN {X 0,Y 389.101,Z 333.866,A -85,B 0,C 180,E1 -11509.168,E2 -11509.168} C_VEL
LIN {X 0,Y 390.511,Z 344.249,A -85,B 0,C 180,E1 -11509.764,E2 -11509.764} C_VEL
LIN {X 0,Y 390.985,Z 349.917,A -85,B 0,C 180,E1 -11510.169,E2 -11510.169} C_VEL
LIN {X 0,Y 390.602,Z 360.273,A -85,B 0,C 180,E1 -11511.074,E2 -11511.074} C_VEL
LIN {X 0,Y 390.222,Z 369.469,A -85,B 0,C 180,E1 -11512.125,E2 -11512.125} C_VEL
LIN {X 0,Y 389.969,Z 377.284,A -85,B 0,C 180,E1 -11513.274,E2 -11513.274} C_VEL
LIN {X 0,Y 389.783,Z 384.117,A -85,B 0,C 180,E1 -11514.57,E2 -11514.57} C_VEL
LIN {X 0,Y 389.505,Z 389.325,A -85,B 0,C 180,E1 -11515.863,E2 -11515.863} C_VEL
LIN {X 0,Y 389.288,Z 392.536,A -85,B 0,C 180,E1 -11516.897,E2 -11516.897} C_VEL
LIN {X 0,Y 389.187,Z 394.963,A -85,B 0,C 180,E1 -11517.932,E2 -11517.932} C_VEL
LIN {X 0,Y 389.091,Z 396.674,A -85,B 0,C 180,E1 -11518.966,E2 -11518.966} C_VEL
LIN {X 0,Y 389.084,Z 397.705,A -85,B 0,C 180,E1 -11520.001,E2 -11520.001} C_VEL
LIN {X 0,Y 389.145,Z 398.066,A -85,B 0,C 180,E1 -11521.036,E2 -11521.036} C_VEL
LIN {X 0,Y 389.271,Z 397.766,A -85,B 0,C 180,E1 -11522.071,E2 -11522.071} C_VEL
LIN {X 0,Y 389.48,Z 396.806,A -85,B 0,C 180,E1 -11523.104,E2 -11523.104} C_VEL
LIN {X 0,Y 390.135,Z 394.058,A -85,B 0,C 180,E1 -11524.651,E2 -11524.651} C_VEL
LIN {X 0,Y 390.427,Z 391.351,A -85,B 0,C 180,E1 -11525.683,E2 -11525.683} C_VEL
LIN {X 0,Y 391.076,Z 385.779,A -85,B 0,C 180,E1 -11527.228,E2 -11527.228} C_VEL
LIN {X 0,Y 391.758,Z 379.531,A -85,B 0,C 180,E1 -11528.512,E2 -11528.512} C_VEL
LIN {X 0,Y 392.425,Z 373.177,A -85,B 0,C 180,E1 -11529.537,E2 -11529.537} C_VEL
LIN {X 0,Y 393.232,Z 365.047,A -85,B 0,C 180,E1 -11530.584,E2 -11530.584} C_VEL
LIN {X 0,Y 393.928,Z 355.202,A -85,B 0,C 180,E1 -11531.58,E2 -11531.58} C_VEL
LIN {X 0,Y 392.069,Z 345.067,A -85,B 0,C 180,E1 -11532.525,E2 -11532.525} C_VEL
LIN {X 0,Y 390.202,Z 337.81,A -85,B 0,C 180,E1 -11533.138,E2 -11533.138} C_VEL
LIN {X 0,Y 390.506,Z 331.817,A -85,B 0,C 180,E1 -11536.737,E2 -11536.737} C_VEL
LIN {X 0,Y 390.917,Z 326.651,A -85,B 0,C 180,E1 -11539.975,E2 -11539.975} C_VEL
LIN {X 0,Y 391.438,Z 321.668,A -85,B 0,C 180,E1 -11543.267,E2 -11543.267} C_VEL
LIN {X 0,Y 392.054,Z 316.955,A -85,B 0,C 180,E1 -11546.626,E2 -11546.626} C_VEL
LIN {X 0,Y 392.563,Z 314.008,A -85,B 0,C 180,E1 -11548.907,E2 -11548.907} C_VEL
LIN {X 0,Y 392.784,Z 311.247,A -85,B 0,C 180,E1 -11551.259,E2 -11551.259} C_VEL
LIN {X 0,Y 392.706,Z 308.903,A -85,B 0,C 180,E1 -11553.697,E2 -11553.697} C_VEL
LIN {X 0,Y 392.476,Z 306.891,A -85,B 0,C 180,E1 -11556.311,E2 -11556.311} C_VEL
LIN {X 0,Y 392.251,Z 305.543,A -85,B 0,C 180,E1 -11558.838,E2 -11558.838} C_VEL
LIN {X 0,Y 392.18,Z 304.851,A -85,B 0,C 180,E1 -11561.534,E2 -11561.534} C_VEL
LIN {X 0,Y 392.269,Z 305.047,A -85,B 0,C 180,E1 -11564.327,E2 -11564.327} C_VEL
LIN {X 0,Y 392.645,Z 306.27,A -85,B 0,C 180,E1 -11567.213,E2 -11567.213} C_VEL
LIN {X 0,Y 393.293,Z 308.781,A -85,B 0,C 180,E1 -11570.211,E2 -11570.211} C_VEL
LIN {X 0,Y 394.019,Z 311.846,A -85,B 0,C 180,E1 -11572.667,E2 -11572.667} C_VEL
LIN {X 0,Y 395.031,Z 316.087,A -85,B 0,C 180,E1 -11575.298,E2 -11575.298} C_VEL
LIN {X 0,Y 396.106,Z 321.105,A -85,B 0,C 180,E1 -11577.84,E2 -11577.84} C_VEL
LIN {X 0,Y 396.687,Z 325.44,A -85,B 0,C 180,E1 -11579.673,E2 -11579.673} C_VEL
LIN {X 0,Y 396.206,Z 328.724,A -85,B 0,C 180,E1 -11580.817,E2 -11580.817} C_VEL
LIN {X 0,Y 394.053,Z 338.816,A -85,B 0,C 180,E1 -11584.09,E2 -11584.09} C_VEL
LIN {X 0,Y 392.213,Z 351.759,A -85,B 0,C 180,E1 -11587.896,E2 -11587.896} C_VEL
LIN {X 0,Y 390.861,Z 365.085,A -85,B 0,C 180,E1 -11591.502,E2 -11591.502} C_VEL
LIN {X 0,Y 392.975,Z 378.205,A -85,B 0,C 180,E1 -11592.109,E2 -11592.109} C_VEL
LIN {X 0,Y 393.684,Z 389.731,A -85,B 0,C 180,E1 -11592.748,E2 -11592.748} C_VEL
LIN {X 0,Y 393.596,Z 399.441,A -85,B 0,C 180,E1 -11593.4,E2 -11593.4} C_VEL
LIN {X 0,Y 392.622,Z 410.57,A -85,B 0,C 180,E1 -11594.292,E2 -11594.292} C_VEL
LIN {X 0,Y 391.602,Z 421.913,A -85,B 0,C 180,E1 -11595.448,E2 -11595.448} C_VEL
LIN {X 0,Y 390.794,Z 432.032,A -85,B 0,C 180,E1 -11596.744,E2 -11596.744} C_VEL
LIN {X 0,Y 390.062,Z 440.321,A -85,B 0,C 180,E1 -11598.041,E2 -11598.041} C_VEL
LIN {X 0,Y 389.404,Z 448.468,A -85,B 0,C 180,E1 -11599.602,E2 -11599.602} C_VEL
LIN {X 0,Y 389.136,Z 454.997,A -85,B 0,C 180,E1 -11601.169,E2 -11601.169} C_VEL
LIN {X 0,Y 389.017,Z 460.188,A -85,B 0,C 180,E1 -11602.735,E2 -11602.735} C_VEL
LIN {X 0,Y 388.914,Z 464.198,A -85,B 0,C 180,E1 -11604.296,E2 -11604.296} C_VEL
LIN {X 0,Y 388.926,Z 467.13,A -85,B 0,C 180,E1 -11605.855,E2 -11605.855} C_VEL
LIN {X 0,Y 389.062,Z 468.536,A -85,B 0,C 180,E1 -11606.893,E2 -11606.893} C_VEL
LIN {X 0,Y 389.123,Z 469.497,A -85,B 0,C 180,E1 -11607.93,E2 -11607.93} C_VEL
LIN {X 0,Y 389.029,Z 469.977,A -85,B 0,C 180,E1 -11608.965,E2 -11608.965} C_VEL
LIN {X 0,Y 389.006,Z 470.053,A -85,B 0,C 180,E1 -11610,E2 -11610} C_VEL
LIN {X 0,Y 389.028,Z 469.71,A -85,B 0,C 180,E1 -11611.035,E2 -11611.035} C_VEL
LIN {X 0,Y 389.134,Z 468.898,A -85,B 0,C 180,E1 -11612.07,E2 -11612.07} C_VEL
LIN {X 0,Y 389.134,Z 467.65,A -85,B 0,C 180,E1 -11613.106,E2 -11613.106} C_VEL
LIN {X 0,Y 388.97,Z 464.88,A -85,B 0,C 180,E1 -11614.664,E2 -11614.664} C_VEL
LIN {X 0,Y 389.033,Z 461.012,A -85,B 0,C 180,E1 -11616.223,E2 -11616.223} C_VEL
LIN {X 0,Y 389.097,Z 454.869,A -85,B 0,C 180,E1 -11618.047,E2 -11618.047} C_VEL
LIN {X 0,Y 389.286,Z 448.052,A -85,B 0,C 180,E1 -11619.613,E2 -11619.613} C_VEL
LIN {X 0,Y 389.594,Z 441.028,A -85,B 0,C 180,E1 -11620.919,E2 -11620.919} C_VEL
LIN {X 0,Y 389.999,Z 432.44,A -85,B 0,C 180,E1 -11622.225,E2 -11622.225} C_VEL
LIN {X 0,Y 390.59,Z 424.155,A -85,B 0,C 180,E1 -11623.263,E2 -11623.263} C_VEL
LIN {X 0,Y 391.121,Z 413.991,A -85,B 0,C 180,E1 -11624.306,E2 -11624.306} C_VEL
LIN {X 0,Y 391.698,Z 402.943,A -85,B 0,C 180,E1 -11625.213,E2 -11625.213} C_VEL
LIN {X 0,Y 392.127,Z 392.86,A -85,B 0,C 180,E1 -11625.862,E2 -11625.862} C_VEL
LIN {X 0,Y 391.207,Z 380.401,A -85,B 0,C 180,E1 -11626.487,E2 -11626.487} C_VEL
LIN {X 0,Y 390.174,Z 367.701,A -85,B 0,C 180,E1 -11626.921,E2 -11626.921} C_VEL
LIN {X 0,Y 390.124,Z 366.498,A -85,B 0,C 180,E1 -11626.98,E2 -11626.98} C_VEL
LIN {X 0,Y 391.158,Z 351.395,A -85,B 0,C 180,E1 -11630.884,E2 -11630.884} C_VEL
LIN {X 0,Y 392.369,Z 338.248,A -85,B 0,C 180,E1 -11634.329,E2 -11634.329} C_VEL
LIN {X 0,Y 393.593,Z 327.697,A -85,B 0,C 180,E1 -11637.119,E2 -11637.119} C_VEL
LIN {X 0,Y 394.644,Z 318.879,A -85,B 0,C 180,E1 -11639.488,E2 -11639.488} C_VEL
LIN {X 0,Y 393.683,Z 313.053,A -85,B 0,C 180,E1 -11641.179,E2 -11641.179} C_VEL
LIN {X 0,Y 390.972,Z 300.135,A -85,B 0,C 180,E1 -11645.115,E2 -11645.115} C_VEL
LIN {X 0,Y 390.076,Z 295.898,A -85,B 0,C 180,E1 -11646.482,E2 -11646.482} C_VEL
LIN {X 0,Y 390.075,Z 295.896,A -85,B 0,C 180,E1 -11649.218,E2 -11649.218} C_VEL
LIN {X 0,Y 390.048,Z 295.902,A -85,B 0,C 180,E1 -11652.374,E2 -11652.374} C_VEL
LIN {X 0,Y 390.05,Z 295.899,A -85,B 0,C 180,E1 -11655.354,E2 -11655.354} C_VEL
LIN {X 0,Y 390.036,Z 295.9,A -85,B 0,C 180,E1 -11658.186,E2 -11658.186} C_VEL
LIN {X 0,Y 390.096,Z 295.894,A -85,B 0,C 180,E1 -11660.907,E2 -11660.907} C_VEL
LIN {X 0,Y 390.09,Z 295.896,A -85,B 0,C 180,E1 -11664.792,E2 -11664.792} C_VEL
LIN {X 0,Y 390.048,Z 295.977,A -85,B 0,C 180,E1 -11667.451,E2 -11667.451} C_VEL
LIN {X 0,Y 391.154,Z 301.141,A -85,B 0,C 180,E1 -11669.794,E2 -11669.794} C_VEL
LIN {X 0,Y 391.426,Z 305.314,A -85,B 0,C 180,E1 -11671.617,E2 -11671.617} C_VEL
LIN {X 0,Y 391.109,Z 313.251,A -85,B 0,C 180,E1 -11675.02,E2 -11675.02} C_VEL
LIN {X 0,Y 390.959,Z 320.898,A -85,B 0,C 180,E1 -11678.375,E2 -11678.375} C_VEL
LIN {X 0,Y 390.756,Z 328.294,A -85,B 0,C 180,E1 -11681.653,E2 -11681.653} C_VEL
LIN {X 0,Y 390.603,Z 335.485,A -85,B 0,C 180,E1 -11684.876,E2 -11684.876} C_VEL
LIN {X 0,Y 390.539,Z 342.526,A -85,B 0,C 180,E1 -11688.055,E2 -11688.055} C_VEL
LIN {X 0,Y 390.517,Z 343.461,A -85,B 0,C 180,E1 -11688.482,E2 -11688.482} C_VEL
LIN {X 0,Y 392.379,Z 351.4,A -85,B 0,C 180,E1 -11689.028,E2 -11689.028} C_VEL
LIN {X 0,Y 392.581,Z 356.76,A -85,B 0,C 180,E1 -11689.425,E2 -11689.425} C_VEL
LIN {X 0,Y 392.183,Z 364.428,A -85,B 0,C 180,E1 -11690.106,E2 -11690.106} C_VEL
LIN {X 0,Y 391.587,Z 372.402,A -85,B 0,C 180,E1 -11691.002,E2 -11691.002} C_VEL
LIN {X 0,Y 391.163,Z 379.083,A -85,B 0,C 180,E1 -11691.995,E2 -11691.995} C_VEL
LIN {X 0,Y 390.872,Z 384.6,A -85,B 0,C 180,E1 -11693.028,E2 -11693.028} C_VEL
LIN {X 0,Y 390.504,Z 387.934,A -85,B 0,C 180,E1 -11693.8,E2 -11693.8} C_VEL
LIN {X 0,Y 390.167,Z 391.495,A -85,B 0,C 180,E1 -11694.831,E2 -11694.831} C_VEL
LIN {X 0,Y 389.809,Z 394.158,A -85,B 0,C 180,E1 -11695.863,E2 -11695.863} C_VEL
LIN {X 0,Y 389.442,Z 396.054,A -85,B 0,C 180,E1 -11696.895,E2 -11696.895} C_VEL
LIN {X 0,Y 389.234,Z 397.218,A -85,B 0,C 180,E1 -11697.929,E2 -11697.929} C_VEL
LIN {X 0,Y 389.117,Z 397.685,A -85,B 0,C 180,E1 -11698.964,E2 -11698.964} C_VEL
LIN {X 0,Y 389.065,Z 397.467,A -85,B 0,C 180,E1 -11699.999,E2 -11699.999} C_VEL
LIN {X 0,Y 389.079,Z 396.561,A -85,B 0,C 180,E1 -11701.034,E2 -11701.034} C_VEL
LIN {X 0,Y 389.185,Z 394.955,A -85,B 0,C 180,E1 -11702.068,E2 -11702.068} C_VEL
LIN {X 0,Y 389.274,Z 392.611,A -85,B 0,C 180,E1 -11703.103,E2 -11703.103} C_VEL
LIN {X 0,Y 389.491,Z 389.411,A -85,B 0,C 180,E1 -11704.138,E2 -11704.138} C_VEL
LIN {X 0,Y 389.743,Z 384.068,A -85,B 0,C 180,E1 -11705.431,E2 -11705.431} C_VEL
LIN {X 0,Y 389.869,Z 378.553,A -85,B 0,C 180,E1 -11706.468,E2 -11706.468} C_VEL
LIN {X 0,Y 390.023,Z 370.24,A -85,B 0,C 180,E1 -11707.661,E2 -11707.661} C_VEL
LIN {X 0,Y 390.307,Z 362.09,A -85,B 0,C 180,E1 -11708.542,E2 -11708.542} C_VEL
LIN {X 0,Y 390.543,Z 352.678,A -85,B 0,C 180,E1 -11709.319,E2 -11709.319} C_VEL
LIN {X 0,Y 390.361,Z 346.372,A -85,B 0,C 180,E1 -11709.716,E2 -11709.716} C_VEL
LIN {X 0,Y 389.571,Z 340.146,A -85,B 0,C 180,E1 -11710.064,E2 -11710.064} C_VEL
LIN {X 0,Y 389.631,Z 332.083,A -85,B 0,C 180,E1 -11713.56,E2 -11713.56} C_VEL
LIN {X 0,Y 389.672,Z 324.081,A -85,B 0,C 180,E1 -11717.08,E2 -11717.08} C_VEL
LIN {X 0,Y 389.786,Z 316.678,A -85,B 0,C 180,E1 -11720.35,E2 -11720.35} C_VEL
LIN {X 0,Y 389.909,Z 307.381,A -85,B 0,C 180,E1 -11724.49,E2 -11724.49} C_VEL
LIN {X 0,Y 390.001,Z 299.661,A -85,B 0,C 180,E1 -11727.937,E2 -11727.937} C_VEL
LIN {X 0,Y 390.135,Z 295.888,A -85,B 0,C 180,E1 -11729.694,E2 -11729.694} C_VEL
LIN {X 0,Y 390.056,Z 295.895,A -85,B 0,C 180,E1 -11733.954,E2 -11733.954} C_VEL
LIN {X 0,Y 390.049,Z 295.896,A -85,B 0,C 180,E1 -11736.482,E2 -11736.482} C_VEL
LIN {X 0,Y 390.032,Z 295.902,A -85,B 0,C 180,E1 -11739.211,E2 -11739.211} C_VEL
LIN {X 0,Y 390.029,Z 295.9,A -85,B 0,C 180,E1 -11742.372,E2 -11742.372} C_VEL
LIN {X 0,Y 390.037,Z 295.9,A -85,B 0,C 180,E1 -11745.353,E2 -11745.353} C_VEL
LIN {X 0,Y 390.023,Z 295.901,A -85,B 0,C 180,E1 -11748.185,E2 -11748.185} C_VEL
LIN {X 0,Y 390.084,Z 295.895,A -85,B 0,C 180,E1 -11750.907,E2 -11750.907} C_VEL
LIN {X 0,Y 390.077,Z 295.896,A -85,B 0,C 180,E1 -11754.792,E2 -11754.792} C_VEL
LIN {X 0,Y 390.02,Z 295.904,A -85,B 0,C 180,E1 -11758.495,E2 -11758.495} C_VEL
LIN {X 0,Y 390.107,Z 295.892,A -85,B 0,C 180,E1 -11762.069,E2 -11762.069} C_VEL
LIN {X 0,Y 390.069,Z 295.895,A -85,B 0,C 180,E1 -11765.518,E2 -11765.518} C_VEL
LIN {X 0,Y 390.044,Z 295.9,A -85,B 0,C 180,E1 -11768.877,E2 -11768.877} C_VEL
LIN {X 0,Y 390.116,Z 295.891,A -85,B 0,C 180,E1 -11772.166,E2 -11772.166} C_VEL
LIN {X 0,Y 390.132,Z 295.887,A -85,B 0,C 180,E1 -11775.392,E2 -11775.392} C_VEL
LIN {X 0,Y 390.135,Z 295.889,A -85,B 0,C 180,E1 -11778.571,E2 -11778.571} C_VEL
LIN {X 0,Y 390.244,Z 295.876,A -85,B 0,C 180,E1 -11782.086,E2 -11782.086} C_VEL
LIN {X 0,Y 390.197,Z 295.878,A -85,B 0,C 180,E1 -11784.833,E2 -11784.833} C_VEL
LIN {X 0,Y 390.394,Z 295.857,A -85,B 0,C 180,E1 -11787.937,E2 -11787.937} C_VEL
LIN {X 0,Y 390.275,Z 295.867,A -85,B 0,C 180,E1 -11791.032,E2 -11791.032} C_VEL
LIN {X 0,Y 390.25,Z 295.871,A -85,B 0,C 180,E1 -11793.097,E2 -11793.097} C_VEL
LIN {X 0,Y 390.274,Z 295.87,A -85,B 0,C 180,E1 -11796.203,E2 -11796.203} C_VEL
LIN {X 0,Y 390.18,Z 295.882,A -85,B 0,C 180,E1 -11799.329,E2 -11799.329} C_VEL
LIN {X 0,Y 390.158,Z 295.884,A -85,B 0,C 180,E1 -11802.484,E2 -11802.484} C_VEL
LIN {X 0,Y 390.127,Z 295.89,A -85,B 0,C 180,E1 -11805.677,E2 -11805.677} C_VEL
LIN {X 0,Y 390.094,Z 295.892,A -85,B 0,C 180,E1 -11808.923,E2 -11808.923} C_VEL
LIN {X 0,Y 390.029,Z 295.901,A -85,B 0,C 180,E1 -11812.235,E2 -11812.235} C_VEL
LIN {X 0,Y 390.109,Z 295.893,A -85,B 0,C 180,E1 -11815.744,E2 -11815.744} C_VEL
LIN {X 0,Y 390.056,Z 295.899,A -85,B 0,C 180,E1 -11819.11,E2 -11819.11} C_VEL
LIN {X 0,Y 390.036,Z 295.899,A -85,B 0,C 180,E1 -11819.968,E2 -11819.968} C_VEL
LIN {X 0,Y 389.392,Z 295.981,A -85,B 0,C 180,E1 -11820.83,E2 -11820.83} C_VEL
LIN {X 0,Y 386.543,Z 296.334,A -85,B 0,C 180,E1 -11822.23,E2 -11822.23} C_VEL
LIN {X 0,Y 384.122,Z 296.639,A -85,B 0,C 180,E1 -11823.362,E2 -11823.362} C_VEL
LIN {X 0,Y 383.088,Z 296.765,A -85,B 0,C 180,E1 -11824.237,E2 -11824.237} C_VEL
LIN {X 0,Y 383.007,Z 296.775,A -85,B 0,C 180,E1 -11824.534,E2 -11824.534} C_VEL
LIN {X 0,Y 382.993,Z 296.776,A -85,B 0,C 180,E1 -11827.905,E2 -11827.905} C_VEL
LIN {X 0,Y 382.976,Z 296.782,A -85,B 0,C 180,E1 -11831.349,E2 -11831.349} C_VEL
LIN {X 0,Y 382.988,Z 296.777,A -85,B 0,C 180,E1 -11834.305,E2 -11834.305} C_VEL
LIN {X 0,Y 383.003,Z 296.777,A -85,B 0,C 180,E1 -11837.242,E2 -11837.242} C_VEL
LIN {X 0,Y 382.979,Z 296.778,A -85,B 0,C 180,E1 -11840.42,E2 -11840.42} C_VEL
LIN {X 0,Y 383.017,Z 296.772,A -85,B 0,C 180,E1 -11844.046,E2 -11844.046} C_VEL
LIN {X 0,Y 383.06,Z 296.766,A -85,B 0,C 180,E1 -11847.857,E2 -11847.857} C_VEL
LIN {X 0,Y 383.202,Z 296.828,A -85,B 0,C 180,E1 -11848.95,E2 -11848.95} C_VEL
LIN {X 0,Y 383.282,Z 300.291,A -85,B 0,C 180,E1 -11850.93,E2 -11850.93} C_VEL
LIN {X 0,Y 382.924,Z 305.924,A -85,B 0,C 180,E1 -11854.07,E2 -11854.07} C_VEL
LIN {X 0,Y 382.642,Z 312.864,A -85,B 0,C 180,E1 -11857.883,E2 -11857.883} C_VEL
LIN {X 0,Y 382.431,Z 319.107,A -85,B 0,C 180,E1 -11861.242,E2 -11861.242} C_VEL
LIN {X 0,Y 382.224,Z 325.344,A -85,B 0,C 180,E1 -11864.539,E2 -11864.539} C_VEL
LIN {X 0,Y 382.129,Z 331.588,A -85,B 0,C 180,E1 -11867.791,E2 -11867.791} C_VEL
LIN {X 0,Y 382.05,Z 333.95,A -85,B 0,C 180,E1 -11868.999,E2 -11868.999} C_VEL
LIN {X 0,Y 383.58,Z 345.706,A -85,B 0,C 180,E1 -11869.711,E2 -11869.711} C_VEL
LIN {X 0,Y 383.944,Z 351.186,A -85,B 0,C 180,E1 -11870.12,E2 -11870.12} C_VEL
LIN {X 0,Y 383.533,Z 361.363,A -85,B 0,C 180,E1 -11871.041,E2 -11871.041} C_VEL
LIN {X 0,Y 383.17,Z 370.2,A -85,B 0,C 180,E1 -11872.079,E2 -11872.079} C_VEL
LIN {X 0,Y 382.933,Z 377.395,A -85,B 0,C 180,E1 -11873.15,E2 -11873.15} C_VEL
LIN {X 0,Y 382.713,Z 384.337,A -85,B 0,C 180,E1 -11874.469,E2 -11874.469} C_VEL
LIN {X 0,Y 382.442,Z 389.649,A -85,B 0,C 180,E1 -11875.786,E2 -11875.786} C_VEL
LIN {X 0,Y 382.229,Z 392.929,A -85,B 0,C 180,E1 -11876.839,E2 -11876.839} C_VEL
LIN {X 0,Y 382.11,Z 395.44,A -85,B 0,C 180,E1 -11877.893,E2 -11877.893} C_VEL
LIN {X 0,Y 382.038,Z 397.235,A -85,B 0,C 180,E1 -11878.947,E2 -11878.947} C_VEL
LIN {X 0,Y 382.027,Z 398.349,A -85,B 0,C 180,E1 -11880.001,E2 -11880.001} C_VEL
LIN {X 0,Y 382.089,Z 398.794,A -85,B 0,C 180,E1 -11881.055,E2 -11881.055} C_VEL
LIN {X 0,Y 382.223,Z 398.576,A -85,B 0,C 180,E1 -11882.109,E2 -11882.109} C_VEL
LIN {X 0,Y 382.447,Z 397.695,A -85,B 0,C 180,E1 -11883.162,E2 -11883.162} C_VEL
LIN {X 0,Y 383.129,Z 395.083,A -85,B 0,C 180,E1 -11884.736,E2 -11884.736} C_VEL
LIN {X 0,Y 383.654,Z 390.909,A -85,B 0,C 180,E1 -11886.312,E2 -11886.312} C_VEL
LIN {X 0,Y 384.464,Z 384.883,A -85,B 0,C 180,E1 -11887.881,E2 -11887.881} C_VEL
LIN {X 0,Y 385.2,Z 378.159,A -85,B 0,C 180,E1 -11889.188,E2 -11889.188} C_VEL
LIN {X 0,Y 386.083,Z 370.706,A -85,B 0,C 180,E1 -11890.307,E2 -11890.307} C_VEL
LIN {X 0,Y 386.932,Z 361.626,A -85,B 0,C 180,E1 -11891.393,E2 -11891.393} C_VEL
LIN {X 0,Y 387.264,Z 356.383,A -85,B 0,C 180,E1 -11891.915,E2 -11891.915} C_VEL
LIN {X 0,Y 385.603,Z 347.271,A -85,B 0,C 180,E1 -11892.821,E2 -11892.821} C_VEL
LIN {X 0,Y 383.23,Z 338.366,A -85,B 0,C 180,E1 -11893.599,E2 -11893.599} C_VEL
LIN {X 0,Y 383.584,Z 332.752,A -85,B 0,C 180,E1 -11897.048,E2 -11897.048} C_VEL
LIN {X 0,Y 384.203,Z 326.501,A -85,B 0,C 180,E1 -11901.106,E2 -11901.106} C_VEL
LIN {X 0,Y 384.796,Z 321.175,A -85,B 0,C 180,E1 -11904.841,E2 -11904.841} C_VEL
LIN {X 0,Y 385.587,Z 316.682,A -85,B 0,C 180,E1 -11908.289,E2 -11908.289} C_VEL
LIN {X 0,Y 385.975,Z 313.379,A -85,B 0,C 180,E1 -11911.152,E2 -11911.152} C_VEL
LIN {X 0,Y 385.912,Z 310.476,A -85,B 0,C 180,E1 -11914.372,E2 -11914.372} C_VEL
LIN {X 0,Y 385.685,Z 308.773,A -85,B 0,C 180,E1 -11916.966,E2 -11916.966} C_VEL
LIN {X 0,Y 385.523,Z 307.576,A -85,B 0,C 180,E1 -11920.035,E2 -11920.035} C_VEL
LIN {X 0,Y 385.554,Z 307.37,A -85,B 0,C 180,E1 -11923.186,E2 -11923.186} C_VEL
LIN {X 0,Y 385.825,Z 308.275,A -85,B 0,C 180,E1 -11926.196,E2 -11926.196} C_VEL
LIN {X 0,Y 386.373,Z 310.301,A -85,B 0,C 180,E1 -11929.093,E2 -11929.093} C_VEL
LIN {X 0,Y 387.16,Z 313.342,A -85,B 0,C 180,E1 -11931.888,E2 -11931.888} C_VEL
LIN {X 0,Y 388.148,Z 317.337,A -85,B 0,C 180,E1 -11934.591,E2 -11934.591} C_VEL
LIN {X 0,Y 389.167,Z 322.088,A -85,B 0,C 180,E1 -11937.195,E2 -11937.195} C_VEL
LIN {X 0,Y 389.864,Z 326.188,A -85,B 0,C 180,E1 -11939.085,E2 -11939.085} C_VEL
LIN {X 0,Y 389.594,Z 329.624,A -85,B 0,C 180,E1 -11940.384,E2 -11940.384} C_VEL
LIN {X 0,Y 387.395,Z 339.276,A -85,B 0,C 180,E1 -11943.61,E2 -11943.61} C_VEL
LIN {X 0,Y 385.403,Z 352.009,A -85,B 0,C 180,E1 -11947.484,E2 -11947.484} C_VEL
LIN {X 0,Y 383.965,Z 364.55,A -85,B 0,C 180,E1 -11951.015,E2 -11951.015} C_VEL
LIN {X 0,Y 386.216,Z 378.004,A -85,B 0,C 180,E1 -11951.69,E2 -11951.69} C_VEL
LIN {X 0,Y 386.974,Z 389.896,A -85,B 0,C 180,E1 -11952.384,E2 -11952.384} C_VEL
LIN {X 0,Y 386.826,Z 400.083,A -85,B 0,C 180,E1 -11953.1,E2 -11953.1} C_VEL
LIN {X 0,Y 385.673,Z 412.248,A -85,B 0,C 180,E1 -11954.137,E2 -11954.137} C_VEL
LIN {X 0,Y 384.62,Z 423.111,A -85,B 0,C 180,E1 -11955.317,E2 -11955.317} C_VEL
LIN {X 0,Y 383.657,Z 433.711,A -85,B 0,C 180,E1 -11956.763,E2 -11956.763} C_VEL
LIN {X 0,Y 382.991,Z 441.592,A -85,B 0,C 180,E1 -11958.086,E2 -11958.086} C_VEL
LIN {X 0,Y 382.309,Z 449.291,A -85,B 0,C 180,E1 -11959.675,E2 -11959.675} C_VEL
LIN {X 0,Y 381.998,Z 456.444,A -85,B 0,C 180,E1 -11961.536,E2 -11961.536} C_VEL
LIN {X 0,Y 381.905,Z 461.159,A -85,B 0,C 180,E1 -11963.13,E2 -11963.13} C_VEL
LIN {X 0,Y 381.862,Z 464.745,A -85,B 0,C 180,E1 -11964.72,E2 -11964.72} C_VEL
LIN {X 0,Y 381.841,Z 466.537,A -85,B 0,C 180,E1 -11965.778,E2 -11965.778} C_VEL
LIN {X 0,Y 381.991,Z 467.92,A -85,B 0,C 180,E1 -11966.836,E2 -11966.836} C_VEL
LIN {X 0,Y 382.055,Z 468.828,A -85,B 0,C 180,E1 -11967.892,E2 -11967.892} C_VEL
LIN {X 0,Y 381.98,Z 469.286,A -85,B 0,C 180,E1 -11968.946,E2 -11968.946} C_VEL
LIN {X 0,Y 381.953,Z 469.338,A -85,B 0,C 180,E1 -11970,E2 -11970} C_VEL
LIN {X 0,Y 381.979,Z 468.941,A -85,B 0,C 180,E1 -11971.054,E2 -11971.054} C_VEL
LIN {X 0,Y 382.086,Z 468.098,A -85,B 0,C 180,E1 -11972.108,E2 -11972.108} C_VEL
LIN {X 0,Y 382.063,Z 466.817,A -85,B 0,C 180,E1 -11973.163,E2 -11973.163} C_VEL
LIN {X 0,Y 381.903,Z 463.98,A -85,B 0,C 180,E1 -11974.75,E2 -11974.75} C_VEL
LIN {X 0,Y 382.008,Z 459.397,A -85,B 0,C 180,E1 -11976.547,E2 -11976.547} C_VEL
LIN {X 0,Y 382.04,Z 453.758,A -85,B 0,C 180,E1 -11978.197,E2 -11978.197} C_VEL
LIN {X 0,Y 382.241,Z 446.831,A -85,B 0,C 180,E1 -11979.792,E2 -11979.792} C_VEL
LIN {X 0,Y 382.691,Z 438.031,A -85,B 0,C 180,E1 -11981.386,E2 -11981.386} C_VEL
LIN {X 0,Y 383.194,Z 428.939,A -85,B 0,C 180,E1 -11982.714,E2 -11982.714} C_VEL
LIN {X 0,Y 383.511,Z 422.962,A -85,B 0,C 180,E1 -11983.445,E2 -11983.445} C_VEL
LIN {X 0,Y 384.174,Z 412.294,A -85,B 0,C 180,E1 -11984.542,E2 -11984.542} C_VEL
LIN {X 0,Y 384.803,Z 400.504,A -85,B 0,C 180,E1 -11985.492,E2 -11985.492} C_VEL
LIN {X 0,Y 385.038,Z 392.222,A -85,B 0,C 180,E1 -11986.026,E2 -11986.026} C_VEL
LIN {X 0,Y 384.065,Z 379.629,A -85,B 0,C 180,E1 -11986.665,E2 -11986.665} C_VEL
LIN {X 0,Y 383.066,Z 366.33,A -85,B 0,C 180,E1 -11987.127,E2 -11987.127} C_VEL
LIN {X 0,Y 384.005,Z 352.771,A -85,B 0,C 180,E1 -11990.717,E2 -11990.717} C_VEL
LIN {X 0,Y 385.239,Z 339.792,A -85,B 0,C 180,E1 -11994.192,E2 -11994.192} C_VEL
LIN {X 0,Y 386.749,Z 327.199,A -85,B 0,C 180,E1 -11997.606,E2 -11997.606} C_VEL
LIN {X 0,Y 387.626,Z 320.281,A -85,B 0,C 180,E1 -11999.507,E2 -11999.507} C_VEL
LIN {X 0,Y 386.935,Z 315.446,A -85,B 0,C 180,E1 -12000.93,E2 -12000.93} C_VEL
LIN {X 0,Y 384.391,Z 303.454,A -85,B 0,C 180,E1 -12004.637,E2 -12004.637} C_VEL
LIN {X 0,Y 383.029,Z 296.775,A -85,B 0,C 180,E1 -12006.835,E2 -12006.835} C_VEL
LIN {X 0,Y 383.014,Z 296.776,A -85,B 0,C 180,E1 -12009.958,E2 -12009.958} C_VEL
LIN {X 0,Y 383.011,Z 296.775,A -85,B 0,C 180,E1 -12012.778,E2 -12012.778} C_VEL
LIN {X 0,Y 383.003,Z 296.779,A -85,B 0,C 180,E1 -12015.789,E2 -12015.789} C_VEL
LIN {X 0,Y 382.994,Z 296.779,A -85,B 0,C 180,E1 -12018.795,E2 -12018.795} C_VEL
LIN {X 0,Y 383.005,Z 296.779,A -85,B 0,C 180,E1 -12022.096,E2 -12022.096} C_VEL
LIN {X 0,Y 383.023,Z 296.778,A -85,B 0,C 180,E1 -12025.331,E2 -12025.331} C_VEL
LIN {X 0,Y 383.027,Z 296.858,A -85,B 0,C 180,E1 -12026.733,E2 -12026.733} C_VEL
LIN {X 0,Y 384.424,Z 303.503,A -85,B 0,C 180,E1 -12029.864,E2 -12029.864} C_VEL
LIN {X 0,Y 384.619,Z 307.471,A -85,B 0,C 180,E1 -12031.634,E2 -12031.634} C_VEL
LIN {X 0,Y 384.237,Z 315.364,A -85,B 0,C 180,E1 -12035.121,E2 -12035.121} C_VEL
LIN {X 0,Y 384.05,Z 322.963,A -85,B 0,C 180,E1 -12038.53,E2 -12038.53} C_VEL
LIN {X 0,Y 383.85,Z 330.498,A -85,B 0,C 180,E1 -12041.864,E2 -12041.864} C_VEL
LIN {X 0,Y 383.674,Z 337.702,A -85,B 0,C 180,E1 -12045.139,E2 -12045.139} C_VEL
LIN {X 0,Y 383.577,Z 344.281,A -85,B 0,C 180,E1 -12048.137,E2 -12048.137} C_VEL
LIN {X 0,Y 385.817,Z 353.899,A -85,B 0,C 180,E1 -12048.839,E2 -12048.839} C_VEL
LIN {X 0,Y 385.614,Z 362.084,A -85,B 0,C 180,E1 -12049.498,E2 -12049.498} C_VEL
LIN {X 0,Y 385.089,Z 370.668,A -85,B 0,C 180,E1 -12050.413,E2 -12050.413} C_VEL
LIN {X 0,Y 384.504,Z 377.468,A -85,B 0,C 180,E1 -12051.333,E2 -12051.333} C_VEL
LIN {X 0,Y 384.124,Z 383.342,A -85,B 0,C 180,E1 -12052.376,E2 -12052.376} C_VEL
LIN {X 0,Y 383.68,Z 388.057,A -85,B 0,C 180,E1 -12053.425,E2 -12053.425} C_VEL
LIN {X 0,Y 383.173,Z 392.529,A -85,B 0,C 180,E1 -12054.737,E2 -12054.737} C_VEL
LIN {X 0,Y 382.791,Z 395.113,A -85,B 0,C 180,E1 -12055.787,E2 -12055.787} C_VEL
LIN {X 0,Y 382.408,Z 396.939,A -85,B 0,C 180,E1 -12056.838,E2 -12056.838} C_VEL
LIN {X 0,Y 382.187,Z 398.032,A -85,B 0,C 180,E1 -12057.891,E2 -12057.891} C_VEL
LIN {X 0,Y 382.063,Z 398.427,A -85,B 0,C 180,E1 -12058.945,E2 -12058.945} C_VEL
LIN {X 0,Y 382.009,Z 398.132,A -85,B 0,C 180,E1 -12059.999,E2 -12059.999} C_VEL
LIN {X 0,Y 382.027,Z 397.148,A -85,B 0,C 180,E1 -12061.053,E2 -12061.053} C_VEL
LIN {X 0,Y 382.108,Z 395.454,A -85,B 0,C 180,E1 -12062.107,E2 -12062.107} C_VEL
LIN {X 0,Y 382.216,Z 392.993,A -85,B 0,C 180,E1 -12063.161,E2 -12063.161} C_VEL
LIN {X 0,Y 382.553,Z 387.708,A -85,B 0,C 180,E1 -12064.741,E2 -12064.741} C_VEL
LIN {X 0,Y 382.668,Z 382.928,A -85,B 0,C 180,E1 -12065.796,E2 -12065.796} C_VEL
LIN {X 0,Y 382.87,Z 376.862,A -85,B 0,C 180,E1 -12066.851,E2 -12066.851} C_VEL
LIN {X 0,Y 382.995,Z 369.59,A -85,B 0,C 180,E1 -12067.856,E2 -12067.856} C_VEL
LIN {X 0,Y 383.29,Z 360.28,A -85,B 0,C 180,E1 -12068.832,E2 -12068.832} C_VEL
LIN {X 0,Y 383.546,Z 350.788,A -85,B 0,C 180,E1 -12069.557,E2 -12069.557} C_VEL
LIN {X 0,Y 383.006,Z 345.032,A -85,B 0,C 180,E1 -12069.904,E2 -12069.904} C_VEL
LIN {X 0,Y 382.517,Z 340.721,A -85,B 0,C 180,E1 -12070.151,E2 -12070.151} C_VEL
LIN {X 0,Y 382.622,Z 333.662,A -85,B 0,C 180,E1 -12073.218,E2 -12073.218} C_VEL
LIN {X 0,Y 382.61,Z 324.583,A -85,B 0,C 180,E1 -12077.221,E2 -12077.221} C_VEL
LIN {X 0,Y 382.733,Z 317.143,A -85,B 0,C 180,E1 -12080.528,E2 -12080.528} C_VEL
LIN {X 0,Y 382.863,Z 308.479,A -85,B 0,C 180,E1 -12084.393,E2 -12084.393} C_VEL
LIN {X 0,Y 382.955,Z 300.975,A -85,B 0,C 180,E1 -12087.778,E2 -12087.778} C_VEL
LIN {X 0,Y 383.089,Z 296.766,A -85,B 0,C 180,E1 -12089.69,E2 -12089.69} C_VEL
